(* CoDeSys 2.3 project: drillMachine_NoPackML.pro *)
(* Title: Use of different IEC-61131-3 languages *)
(* Version: 1.0.0 *)
(* Author: Niko Siltala (TUT) *)
(* Description: Use of different IEC-61131-3 languages to control a lift door. *)
(* Libraries: Util.lib 26.9.14 10:12:46, STANDARD.LIB 16.8.17 14:08:57 *)

(* Global variable list: Global_Variables *)
VAR_GLOBAL
	(*Math constants*)
	MATH 				: CONSTANTS_MATH;		(*Mathematical constants from OSCAT 333*)
	lastRandom			: REAL;		(*Last Random number*)

	(*ConveyourIn - Left*)
	I_ConvIn_PartPresent: BOOL;	(*Sensor: Part is present*)
	O_ConvIn_MotON		: BOOL;	(*Conveyour In: Motor ON*)

	(*ConveyourOut - Right*)
	I_ConvOut_PartPresent: BOOL;(*Sensor: Part is present*)
	O_ConvOut_MotON		: BOOL;	(*Conveyour Out: Motor ON*)

	(*Manipulator - Left*)
	I_ManiL_Limit_Up	: BOOL;	(*Manipulator Left: Limit: Up*)
	I_ManiL_Limit_Dn	: BOOL;	(*Manipulator Left: Limit: Down*)
	I_ManiL_Limit_Home	: BOOL;	(*Manipulator Left: Home sensor*)
	I_ManiL_Turned_Left	: BOOL;	(*Manipulator Left: Turned to left*)
	I_ManiL_Turned_Right: BOOL;	(*Manipulator Left: Turned to right*)
	I_ManiL_Gripper_Open: BOOL;	(*Manipulator Left: Gripper is open*)

	O_ManiL_Turn_Left	: BOOL;	(*Manipulator Left: Turn to left position. Controls the valve*)
	O_ManiL_Turn_Right	: BOOL;	(*Manipulator Left: Turn to right position. Controls the valve*)
	O_ManiL_Gripper_Close: BOOL;(*Manipulator Left: Closes Gripper. Controls the valve*)

	bManiL_axZ_Enable	: BOOL;	(*Manipulator Left: Z-axis: enable*)
	bManiL_axZ_Start	: BOOL;	(*Manipulator Left: Z-axis: Start motion*)
	fManiL_axZ_Velo		: REAL;	(*Manipulator Left: Z-axis: Velocity*)
	fManiL_axZ_TargetPos: REAL;	(*Manipulator Left: Z-axis: Target position*)
	fManiL_axZ_CurrPos	: REAL;	(*Manipulator Left: Z-axis: Current position*)
	bManiL_axZ_InTargetPos	: BOOL;	(*Manipulator Left: Z-axis: Target position is reached*)

	(*Drilling Machine*)
	I_Drill_Limit_Up	: BOOL;	(*Drill: Limit: Up*)
	I_Drill_Limit_Dn	: BOOL;	(*Drill: Limit: Down*)
	I_Drill_Limit_Home	: BOOL;	(*Drill: Home sensor*)
	I_Drill_Fixture_Open: BOOL;	(*Drill: Fixture is open*)
	I_Drill_Fixture_Closed: BOOL;	(*Drill: Fixture is closed*)

	O_Drill_Spindle_On	: BOOL;	(*Drill: Turn on drill spindle.*)
	O_Drill_Fixture_Close: BOOL;(*Drill: Closes Fixture. Controls the valve*)

	bDrill_axZ_Enable	: BOOL;	(*Drill: Z-axis: enable*)
	bDrill_axZ_Start	: BOOL;	(*Drill: Z-axis: Start motion*)
	fDrill_axZ_Velo		: REAL;	(*Drill: Z-axis: Velocity*)
	fDrill_axZ_TargetPos: REAL;	(*Drill: Z-axis: Target position*)
	fDrill_axZ_CurrPos	: REAL;	(*Drill: Z-axis: Current position*)
	bDrill_axZ_InTargetPos	: BOOL;	(*Drill: Z-axis: Target position is reached*)

	(*Manipulator - Right*)
	I_ManiR_Limit_Up	: BOOL;	(*Manipulator Right: Limit: Up*)
	I_ManiR_Limit_Dn	: BOOL;	(*Manipulator Right: Limit: Down*)
	I_ManiR_Limit_Home	: BOOL;	(*Manipulator Right: Home sensor*)
	I_ManiR_Turned_Left	: BOOL;	(*Manipulator Right: Turned to left*)
	I_ManiR_Turned_Right: BOOL;	(*Manipulator Right: Turned to right*)
	I_ManiR_Gripper_Open: BOOL;	(*Manipulator Right: Gripper is open*)

	O_ManiR_Turn_Left	: BOOL;	(*Manipulator Right: Turn to left position. Controls the valve*)
	O_ManiR_Turn_Right	: BOOL;	(*Manipulator Right: Turn to right position. Controls the valve*)
	O_ManiR_Gripper_Close: BOOL;(*Manipulator Right: Closes Gripper. Controls the valve*)

	bManiR_axZ_Enable	: BOOL;	(*Manipulator Right: Z-axis: enable*)
	bManiR_axZ_Start	: BOOL;	(*Manipulator Right: Z-axis: Start motion*)
	fManiR_axZ_Velo		: REAL;	(*Manipulator Right: Z-axis: Velocity*)
	fManiR_axZ_TargetPos: REAL;	(*Manipulator Right: Z-axis: Target position*)
	fManiR_axZ_CurrPos	: REAL;	(*Manipulator Right: Z-axis: Current position*)
	bManiR_axZ_InTargetPos	: BOOL;	(*Manipulator Right: Z-axis: Target position is reached*)


	(*Control panel and indications*)
	I_EmergencyClear	: BOOL;	(*Emergency Circuit is clear*)
	I_Btn_Reset		: BOOL;	(*Button: Reset*)
	I_Btn_Start		: BOOL;	(*Button: Start*)
	I_Btn_Stop		: BOOL;	(*Button: Stop*)

	O_Light_Start	: BOOL;	(*Light: Running*)
	O_Light_Stop	: BOOL;	(*Light: Stopped*)
	O_Beacon_Red	: BOOL;	(*Beacon Light: red*)
	O_Beacon_Yellow	: BOOL;	(*Beacon Light: yellow*)
	O_Beacon_Green	: BOOL;	(*Beacon Light: green*)

(* -------------HMI INPUTS (from HMI to PLC) -------------------*)
	HMI_uModeReq		: UINT :=5;		(*Mode request. DEFAULT:PRODUCTION1*)
(* -------------HMI OUTPUTS (from PLC to HMI) -------------------*)
	PLC_uModeCurrent	: UINT;			(*Current Mode*)
	PLC_uStateCurrent	: UINT;			(*Current State*)

(*-----------------------FUNCTION BLOCKS----------------*)
(*	fbStateModel		: FB_PackMLStateModel_ST;	(*FB for executing PackML state model*) *)
END_VAR

(* Data type *)
TYPE CONSTANTS_MATH :
STRUCT
	PI : REAL := 	3.14159265358979323846264338327950288;		(* Kreiszahl PI *)
	PI2 : REAL := 	6.28318530717958647692528676655900576;	(* PI * 2 *)
	PI4 : REAL :=  12.56637061435917295385057353311801152;	(* PI * 4 *)
	PI05 : REAL :=  1.5707963267949;							(* PI / 2 *)
	PI025 : REAL := 0.785398163397448;							(* PI / 4 *)
	PI_INV : REAL := 0.318309886183791;						(* 1 / PI *)
	E : REAL := 	2.71828182845904523536028747135266249;		(* Euler constant e *)
	E_INV : REAL := 0.367879441171442;							(* 1 / e *)
	SQ2 : REAL :=	1.4142135623731;							(* Wurzel von 2 *)
	FACTS : ARRAY[0..12] OF DINT := 1,1,2,6,24,120,720,5040,40320,362880,3628800,39916800,479001600;
END_STRUCT
END_TYPE



(*
From OSCAT 333
revision history
hm	26.10.2008	rev 1.0
	original version

hm	26. mar. 2011	rev 1.1
	added array facts
*)

(* Data type *)
TYPE ST_Part :
(*Data structure for the simulated parts *)
STRUCT
	bExists		: BOOL;	(* Part exists *)
	bHasHole	: BOOL;	(* Part has hole *)
	posX		: REAL;	(* X-position of the part*)
	posY		: REAL;	(* Y-position of the part*)
END_STRUCT
END_TYPE

(* POU PRG_MAIN, ST *)
(* Main Program for Simulated Drill machine.  Perfoms required co-ordination and calling of function blocks
and connects handshake signals etc.  Mode manager FB is used to handle User inputs via HMI
Author: Nicolas Trimborn, nicolas.trimborn@tuni.fi, TUNI
Date: 2020-02-29
Version: 1.0 *) 

PROGRAM PRG_MAIN
VAR
	(* Function Blocks for Machine *)
	fbSFCExample 		: FB_SFC_Example;
	fbMngr					: FB_SimpleManager;
	fbLights				: FB_Lights;
	fbConveyorLeft		: FB_Conveyor_Left;
	fbConveyorRight		: FB_Conveyor_Right;
	fbManipulatorLeft		: FB_Manipulator;
	fbDrill					: FB_Drill;
	fbManipulatorRight	: FB_Manipulator;


	startTrig				: R_TRIG;	 (* Used to restart system after E_Stop Event *)
	(* Status Flags *)
	bStoppedOkAll		: BOOL := TRUE;
	bAll_InitOK			: BOOL := FALSE;

	(* Flags used to handle E_Stop recovery *)
	bStopRequested		: BOOL := FALSE;
	bE_StopRestart		: BOOL := FALSE;

END_VAR
(* Triggers a restart after emergency is cleared *)
startTrig(CLK:= I_EmergencyClear);
IF bAll_InitOK AND NOT bStopRequested THEN
	bE_StopRestart := startTrig.Q;
ELSE
	bE_StopRestart := FALSE;
END_IF

(* Mode Mangager to Handle HMI Buttons*)
fbMngr(
	bEmergencyClear:= I_EmergencyClear,
	bReset:= I_Btn_Reset,
	bStart:= I_Btn_Start OR bE_StopRestart,
	bStop:= I_Btn_Stop,
	bStopOK_All := bStoppedOkAll,
	oEmergencyClear=>,
	oRun=>,
	oStopRequested => bStopRequested );

(* Controls HMI lights based on system state *)
fbLights(
	bReset:= ,
	I_Emergency:= NOT fbMngr.oEmergencyClear,
	I_Stopped:= bStoppedOkAll AND NOT fbMngr.oRun AND fbMngr.oEmergencyClear ,
	I_Stopping:= fbMngr.oEmergencyClear AND NOT fbMngr.oRun AND NOT bStoppedOkAll,
	I_Starting:=  fbMngr.oRun AND NOT bAll_InitOK,
	I_Executing:=  fbMngr.oRun AND bAll_InitOK,
	I_Suspend:= ,
	I_Error:= (PRG_Simulator.wError_ManipL <> 0) OR (PRG_Simulator.wError_ManipR <> 0) OR (PRG_Simulator.wError_Drill <> 0),

	O_Light_Start=> O_Light_Start ,
	O_Light_Stop=> O_Light_Stop ,
	O_Beacon_Red=> O_Beacon_Red,
	O_Beacon_Yellow=> O_Beacon_Yellow,
	O_Beacon_Green=> O_Beacon_Green );

(*Call emergency actions, if emergency is active, other FB not called as long as
Estop is active *)
IF NOT fbMngr.oEmergencyClear THEN
	actEmergency();
	RETURN;
END_IF

(* Continue running system unless all FB indicate ok to Stop *)
IF fbMngr.oRun OR NOT bStoppedOkAll THEN
	fbConveyorLeft (
		bRun := fbMngr.oRun ,
		I_Reset:= NOT  fbMngr.oEmergencyClear  ,
		O_ConvRunning=> O_ConvIn_MotON,
		I_PartEndSensor:=  I_ConvIn_PartPresent,
		hiPartAvail_FromLeft:= TRUE ,
		hiRdyToReceive_FromRight:= fbManipulatorLeft.hoReadyToRecieve_ToLeft,
		hoPartAvail_toRight=> ,
		hoReadyToRecieve_ToLeft=> );
	
	fbManipulatorLeft(
		I_Enable						:=  fbMngr.oRun,
		I_Reset						:=   ,
		b_LeftManip					:= TRUE ,
		I_Mani_Limit_Up				:= I_ManiL_Limit_Up,
		I_Mani_Limit_Dn				:= I_ManiL_Limit_Dn,
		I_Mani_Limit_Home			:= I_ManiL_Limit_Home ,
		I_Mani_Turned_Left			:= I_ManiL_Turned_Left,
		I_Mani_Turned_Right			:= I_ManiL_Turned_Right ,
		I_Mani_Gripper_Open		:= I_ManiL_Gripper_Open ,
		I_fMani_axZ_CurrPos			:= fManiL_axZ_CurrPos ,
		I_bMani_axZ_InTargetPos	:= bManiL_axZ_InTargetPos,
	
		hiPartAvail_FromLeft			:= fbConveyorLeft.hoPartAvail_ToRight ,
		hiRdyToReceive_FromRight	:= fbDrill.hoReadyToRecieve_ToLeft,
		hoReadyToRecieve_ToLeft	=> ,
		hoPartAvail_ToRight			=> ,

		O_Mani_Turn_Left			=> O_ManiL_Turn_Left ,
		O_Mani_Turn_Right			=> O_ManiL_Turn_Right ,
		O_Mani_Gripper_Close		=> O_ManiL_Gripper_Close ,
		O_bMani_axZ_Enable		=> bManiL_axZ_Enable ,
		O_bMani_axZ_Start			=> bManiL_axZ_Start ,
		O_fMani_axZ_Velo			=> fManiL_axZ_Velo,
		O_fMani_axZ_TargetPos		=> fManiL_axZ_TargetPos );
	
	fbDrill(
		I_Enable						:= fbMngr.oRun,
		I_Reset						:=  ,
		I_Drill_Limit_Up				:= I_Drill_Limit_Up,
		I_Drill_Limit_Dn				:= I_Drill_Limit_Dn ,
		I_Drill_Limit_Home			:= I_Drill_Limit_Home,
		I_Drill_Fixture_Open			:= I_Drill_Fixture_Open,
		I_Drill_Fixture_Closed		:= I_Drill_Fixture_Closed,
		fDrill_axZ_CurrPos			:= fDrill_axZ_CurrPos ,
		bDrill_axZ_InTargetPos		:= bDrill_axZ_InTargetPos ,
	
		hiPartAvail_FromLeft			:= fbManipulatorLeft.hoPartAvail_ToRight ,
		hiRdyToReceive_FromRight	:= fbManipulatorRight.hoReadyToRecieve_ToLeft ,
		hoReadyToRecieve_ToLeft	=> ,
		hoPartAvail_ToRight			=> ,
	
		O_Drill_Spindle_On			=> O_Drill_Spindle_On ,
		O_Drill_Fixture_Close		=> O_Drill_Fixture_Close ,
		bDrill_axZ_Enable			=> bDrill_axZ_Enable ,
		bDrill_axZ_Start				=> bDrill_axZ_Start ,
		fDrill_axZ_Velo				=> fDrill_axZ_Velo,
		fDrill_axZ_TargetPos			=> fDrill_axZ_TargetPos );
	
	fbManipulatorRight(
		I_Enable						:=  fbMngr.oRun,
		I_Reset						:=   ,
		b_LeftManip					:= FALSE ,
		I_Mani_Limit_Up				:= I_ManiR_Limit_Up,
		I_Mani_Limit_Dn				:= I_ManiR_Limit_Dn,
		I_Mani_Limit_Home			:= I_ManiR_Limit_Home ,
		I_Mani_Turned_Left			:= I_ManiR_Turned_Left,
		I_Mani_Turned_Right			:= I_ManiR_Turned_Right ,
		I_Mani_Gripper_Open		:= I_ManiR_Gripper_Open ,
		I_fMani_axZ_CurrPos			:= fManiR_axZ_CurrPos ,
		I_bMani_axZ_InTargetPos	:= bManiR_axZ_InTargetPos,
	
		hiPartAvail_FromLeft			:= fbDrill.hoPartAvail_ToRight,
		hiRdyToReceive_FromRight	:= fbConveyorRight.hoReadyToRecieve_ToLeft,
		hoReadyToRecieve_ToLeft	=> ,
		hoPartAvail_ToRight			=> ,
	
		O_Mani_Turn_Left			=> O_ManiR_Turn_Left ,
		O_Mani_Turn_Right			=> O_ManiR_Turn_Right ,
		O_Mani_Gripper_Close		=> O_ManiR_Gripper_Close ,
		O_bMani_axZ_Enable		=> bManiR_axZ_Enable ,
		O_bMani_axZ_Start			=> bManiR_axZ_Start ,
		O_fMani_axZ_Velo			=> fManiR_axZ_Velo,
		O_fMani_axZ_TargetPos		=> fManiR_axZ_TargetPos );
	
	fbConveyorRight (
		bRun := fbMngr.oRun ,
		I_Reset:=   ,
		O_ConvRunning=> O_ConvOut_MotON,
		I_PartEndSensor:=  I_ConvOut_PartPresent,
	
		hiPartAvail_FromLeft:= fbManipulatorRight.hoPartAvail_ToRight  ,
		hiRdyToReceive_FromRight:= TRUE ,
		hoPartAvail_toRight=> ,
		hoReadyToRecieve_ToLeft=> );
END_IF

(* Continously checks if all FB are OK to Stop *)
IF fbConveyorLeft.bStopOk AND fbManipulatorLeft.bStopOk AND fbManipulatorRight.bStopOk AND fbDrill.bStopOk AND  fbConveyorRight.bStopOk THEN
	bStoppedOkAll := TRUE;
ELSE
	bStoppedOkAll := FALSE;
END_IF

(* Checks if all FB are been initialised *)
IF fbManipulatorLeft.bInitialised AND fbManipulatorRight.bInitialised AND fbDrill.bInitialised THEN
	bAll_InitOK := TRUE;
ELSE
	bAll_InitOK := FALSE;
END_IF
END_PROGRAM
ACTION actEmergency:
(* Emergency action which sets outputs to required safe state *)

(* Conveyors *)
O_ConvIn_MotON					:= FALSE;
O_ConvOut_MotON	 			:= FALSE;

(* Manipulators *)
O_ManiL_Turn_Left		 		:= FALSE;
O_ManiL_Turn_Right		 		:= FALSE;
O_ManiR_Turn_Left		 		:= FALSE;
O_ManiR_Turn_Right		 		:= FALSE;
bManiL_axZ_Start					:= FALSE;
bManiR_axZ_Start				:= FALSE;

(*  Avoid Dropping Objects *)
IF I_ManiL_Gripper_Open THEN
	O_ManiL_Gripper_Close 	:= FALSE;
ELSE
	O_ManiL_Gripper_Close		:= TRUE;
END_IF
(* Drill *)
bDrill_axZ_Start 					:= FALSE;
O_Drill_Spindle_On				:= FALSE;

(*  Avoid Toggling fixture Objects *)
IF I_Drill_Fixture_Open THEN
	O_Drill_Fixture_Close 		:= FALSE;
ELSE
	O_Drill_Fixture_Close		:= TRUE;
END_IF
END_ACTION

(* POU Examples/FB_SFC_Example, SFC *)
FUNCTION_BLOCK FB_SFC_Example
VAR_INPUT
	bReset		: BOOL;	(*Reset Request*)
END_VAR
VAR_OUTPUT
END_VAR
VAR
	bLocalReset	: BOOL;	(*Performs local reset*)
	SFCReset 	: BOOL;	(*Resets the execution of SFC to init once this SFCFlag is set true *)
END_VAR
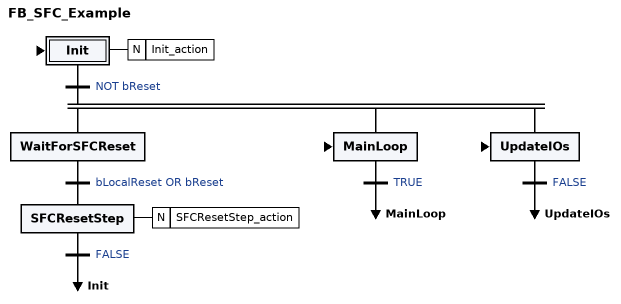
INITIAL_STEP Init:
	Init_action(N);
END_STEP
TRANSITION FROM Init TO (WaitForSFCReset, MainLoop, UpdateIOs) := NOT bReset;
END_TRANSITION
STEP WaitForSFCReset:
END_STEP
TRANSITION FROM WaitForSFCReset TO SFCResetStep := bLocalReset OR bReset;
END_TRANSITION
STEP SFCResetStep:
	SFCResetStep_action(N);
END_STEP
TRANSITION FROM SFCResetStep TO Init := FALSE;
END_TRANSITION
STEP MainLoop:
END_STEP
TRANSITION FROM MainLoop TO MainLoop := TRUE;
END_TRANSITION
STEP UpdateIOs:
END_STEP
TRANSITION FROM UpdateIOs TO UpdateIOs := FALSE;
END_TRANSITION

ACTION Init_action:
SFCReset 	:= FALSE;
bLocalReset	:= FALSE;
END_ACTION

ACTION SFCResetStep_action:
SFCReset := TRUE;
END_ACTION
END_FUNCTION_BLOCK

(* POU FBs/FB_SimpleManager, ST *)
FUNCTION_BLOCK FB_SimpleManager
(*Simple manager following emergency and run/stop state. Outputs can be used to enable user's processes and programs.
Niko Siltala niko.siltala@tuni.fi, 
Tampere University, ENS, ATME.
9.10.2019 v1 *)
VAR_INPUT
	bEmergencyClear		: BOOL;	(*Emergency cleared*)
	bReset				: BOOL;	(*Reset signal*)
	bStart					: BOOL;	(*Start signal*)
	bStop					: BOOL;	(*Stop signal*)
	bStopOK_All			: BOOL;
END_VAR
VAR_OUTPUT
	oEmergencyClear		: BOOL;	(*Emergency is cleared*)
	oRun					: BOOL;	(*System can be started and running*)
	oStopRequested		: BOOL;
END_VAR
VAR
	rsStopRequest		: RS;
	rsEmergency			: RS;
	rsRunning				: RS;
	bResetRequired		: BOOL := TRUE;	(*reset is required*)
END_VAR
(*Defaults*)
(*Reset done*)
IF bReset THEN
	bResetRequired	:= FALSE;
END_IF;

(*Emergency active or cleared?*)
rsEmergency(
	SET:= bReset,
	RESET1:= NOT bEmergencyClear,
	Q1=> oEmergencyClear );

(*Running or stop?*)
rsRunning(
	SET:= bStart,
	RESET1:= (NOT oEmergencyClear) OR bStop OR bResetRequired ,
	Q1=> oRun );

rsStopRequest(
	SET:= bStop,
	RESET1:= bStopOK_All OR bStart,
	Q1=> oStopRequested );
END_FUNCTION_BLOCK

(* POU FBs/FB_Lights, SFC *)
(*Function Block to control the lights of the drill machine based on inputs and functional requirements provided with assignment
Author: Nicolas Trimborn, nicolas.trimborn@tuni.fi, TUNI
Date: 2020-02-29
Version: 1.0 *) 
FUNCTION_BLOCK FB_Lights
VAR_INPUT
	bReset				: BOOL;	(*Reset Request*)
	(* Input States for machine *)
	I_Emergency			: BOOL;
	I_Stopped				: BOOL;
	I_Stopping				: BOOL;
	I_Starting				: BOOL;
	I_Executing			: BOOL;
	I_Suspend			: BOOL;
	I_Error					: BOOL;
END_VAR
VAR_OUTPUT
	(* Light outputs controlled based on input states *)
	O_Light_Start			: BOOL;	(*Light: Running*)
	O_Light_Stop			: BOOL;	(*Light: Stopped*)
	O_Beacon_Red		: BOOL;	(*Beacon Light: red*)
	O_Beacon_Yellow	: BOOL;	(*Beacon Light: yellow*)
	O_Beacon_Green		: BOOL;	(*Beacon Light: greem*)
END_VAR
VAR
	bLocalReset			: BOOL;	(*Performs local reset*)
	SFCReset 			: BOOL;	(*Resets the execution of SFC to init once this SFCFlag is set true *)
 	fbBlinker				: BLINK;     (* Standard Blinker Function Block *)
END_VAR
VAR CONSTANT
	(* 1 Hz Blink requirement *)
	blinkInterval    			: TIME := t#1s;
END_VAR
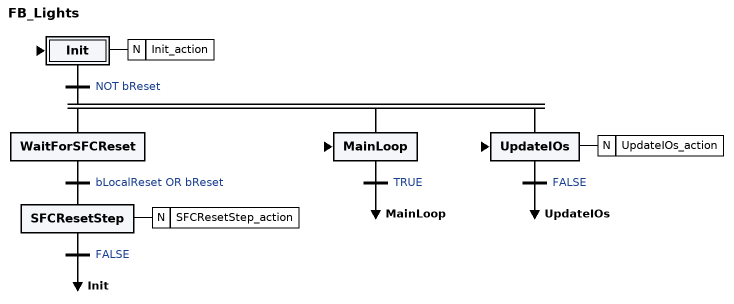
INITIAL_STEP Init:
	Init_action(N);
END_STEP
TRANSITION FROM Init TO (WaitForSFCReset, MainLoop, UpdateIOs) := NOT bReset;
END_TRANSITION
STEP WaitForSFCReset:
END_STEP
TRANSITION FROM WaitForSFCReset TO SFCResetStep := bLocalReset OR bReset;
END_TRANSITION
STEP SFCResetStep:
	SFCResetStep_action(N);
END_STEP
TRANSITION FROM SFCResetStep TO Init := FALSE;
END_TRANSITION
STEP MainLoop:
END_STEP
TRANSITION FROM MainLoop TO MainLoop := TRUE;
END_TRANSITION
STEP UpdateIOs:
	UpdateIOs_action(N);
END_STEP
TRANSITION FROM UpdateIOs TO UpdateIOs := FALSE;
END_TRANSITION

ACTION Init_action:
SFCReset 	:= FALSE;
bLocalReset	:= FALSE;
fbBlinker(ENABLE:= FALSE);
END_ACTION

ACTION SFCResetStep_action:
SFCReset := TRUE;
END_ACTION

ACTION UpdateIOs_action:
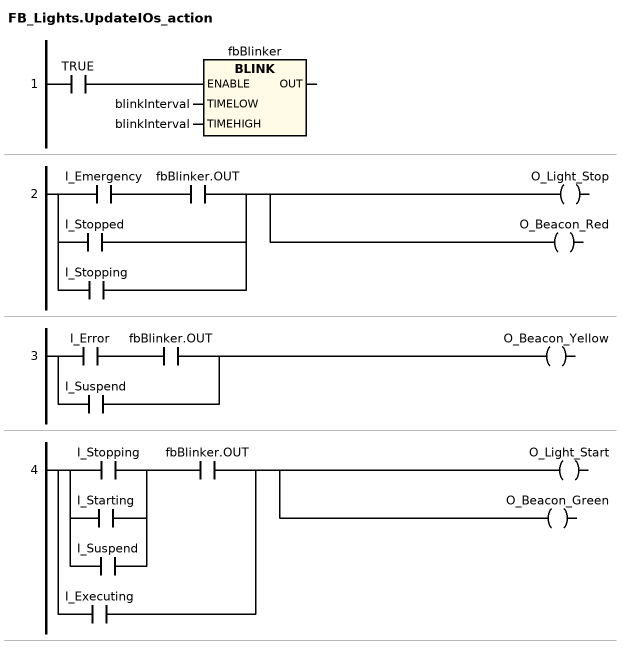
_LD_ (* Ladder Diagram *)
NETWORK 1
	[TRUE] - fbBlinker:BLINK(ENABLE: *, TIMELOW: blinkInterval, TIMEHIGH: blinkInterval)
NETWORK 2
	{ [I_Emergency] - [fbBlinker.OUT] | [I_Stopped] | [I_Stopping] } --- (O_Light_Stop) (O_Beacon_Red)
NETWORK 3
	{ [I_Error] - [fbBlinker.OUT] | [I_Suspend] } --- (O_Beacon_Yellow)
NETWORK 4
	{ { [I_Stopping] | [I_Starting] | [I_Suspend] } - [fbBlinker.OUT] | [I_Executing] } --- (O_Light_Start) (O_Beacon_Green)
_END_LD_
(* the same logic as Structured Text *)
(* Network 1 *)
fbBlinker(ENABLE := TRUE, TIMELOW := blinkInterval, TIMEHIGH := blinkInterval);
(* Network 2 *)
O_Light_Stop := I_Emergency AND fbBlinker.OUT OR I_Stopped OR I_Stopping;
O_Beacon_Red := O_Light_Stop;
(* Network 3 *)
O_Beacon_Yellow := I_Error AND fbBlinker.OUT OR I_Suspend;
(* Network 4 *)
O_Light_Start := (I_Stopping OR I_Starting OR I_Suspend) AND fbBlinker.OUT OR I_Executing;
O_Beacon_Green := O_Light_Start;
END_ACTION
END_FUNCTION_BLOCK

(* POU FBs/FB_Conveyor_Left, SFC *)
(*Function Block to control the left conveyor of simulated drill machine. When bRun is set,
will continously transport added parts to end and notify downstream machine when part is 
availble using SMEMA handshakes.  hiPartAvail_FromLeft always True as this is the start
of production line and assumed to always have parts avalible, but need to be added by operator
Author: Nicolas Trimborn, nicolas.trimborn@tuni.fi, TUNI
Date: 2020-02-29
Version: 1.0 *) 

FUNCTION_BLOCK FB_Conveyor_Left
VAR_INPUT
	bRun		 				: BOOL; 	(*Run Conveyor Function Block*)
	I_Reset		 			: BOOL;	(*Reset Function Block*)
	I_PartEndSensor 			: BOOL;	(*Part End Sensor Input*)

	(* SMEMA Handshake Inputs *)
	hiPartAvail_FromLeft			: BOOL;
	hiRdyToReceive_FromRight	: BOOL;
END_VAR
VAR_OUTPUT
	O_ConvRunning			       : BOOL; (*Output to Simulated conveyor motor*)
	bStopOk						: BOOL; (* bStopOk indicates when there are no parts for processing  and FB is ok to STOP*)

	(* SMEMA Handshake Outputs *)
	hoReadyToRecieve_ToLeft	: BOOL;
	hoPartAvail_ToRight			: BOOL;
END_VAR
VAR
	bLocalReset				: BOOL := FALSE;	(*Performs local reset*)
	SFCReset 				: BOOL := FALSE;	(*Resets the execution of SFC to init once this SFCFlag is set true *)
END_VAR
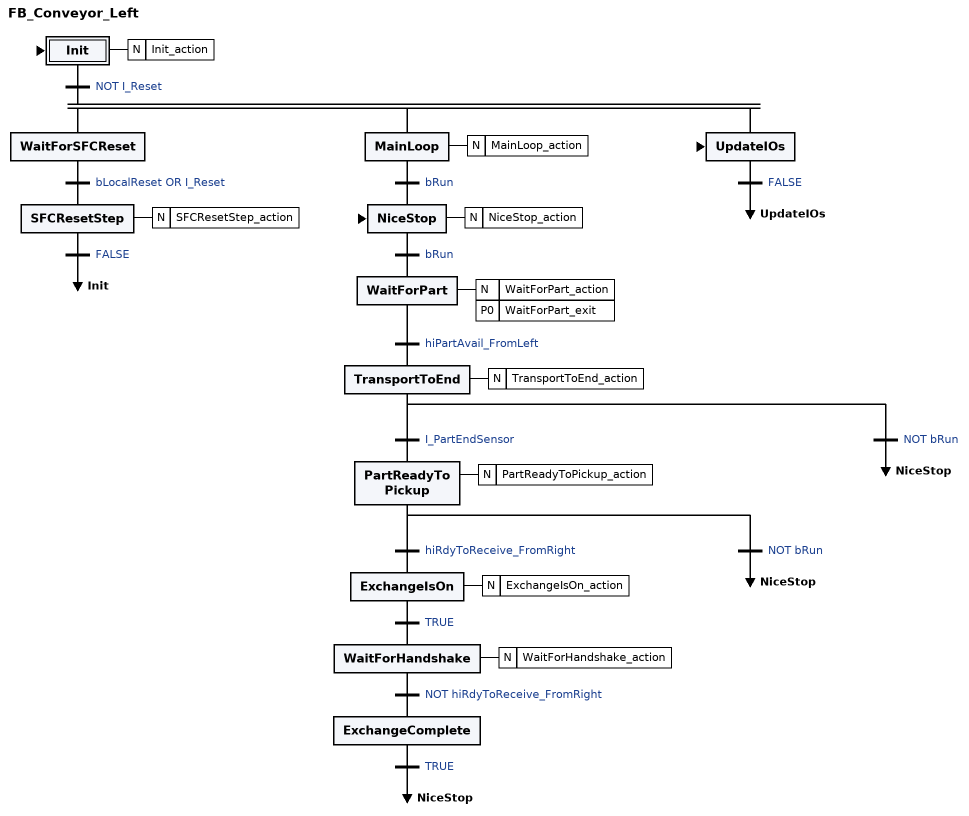
INITIAL_STEP Init:
	Init_action(N);
END_STEP
TRANSITION FROM Init TO (WaitForSFCReset, MainLoop, UpdateIOs) := NOT I_Reset;
END_TRANSITION
STEP WaitForSFCReset:
END_STEP
TRANSITION FROM WaitForSFCReset TO SFCResetStep := bLocalReset OR I_Reset;
END_TRANSITION
STEP MainLoop:
	MainLoop_action(N);
END_STEP
TRANSITION FROM MainLoop TO NiceStop := bRun;
END_TRANSITION
STEP NiceStop:
	NiceStop_action(N);
END_STEP
TRANSITION FROM NiceStop TO WaitForPart := bRun;
END_TRANSITION
STEP WaitForPart:
	WaitForPart_action(N);
	WaitForPart_exit(P0);
END_STEP
TRANSITION FROM WaitForPart TO TransportToEnd := hiPartAvail_FromLeft;
END_TRANSITION
STEP TransportToEnd:
	TransportToEnd_action(N);
END_STEP
TRANSITION FROM TransportToEnd TO PartReadyToPickup := I_PartEndSensor;
END_TRANSITION
TRANSITION FROM TransportToEnd TO NiceStop := NOT bRun;
END_TRANSITION
STEP PartReadyToPickup:
	PartReadyToPickup_action(N);
END_STEP
TRANSITION FROM PartReadyToPickup TO ExchangeIsOn := hiRdyToReceive_FromRight;
END_TRANSITION
TRANSITION FROM PartReadyToPickup TO NiceStop := NOT bRun;
END_TRANSITION
STEP ExchangeIsOn:
	ExchangeIsOn_action(N);
END_STEP
TRANSITION FROM ExchangeIsOn TO WaitForHandshake := TRUE;
END_TRANSITION
STEP WaitForHandshake:
	WaitForHandshake_action(N);
END_STEP
TRANSITION FROM WaitForHandshake TO ExchangeComplete := NOT hiRdyToReceive_FromRight;
END_TRANSITION
STEP ExchangeComplete:
END_STEP
TRANSITION FROM ExchangeComplete TO NiceStop := TRUE;
END_TRANSITION
STEP UpdateIOs:
END_STEP
TRANSITION FROM UpdateIOs TO UpdateIOs := FALSE;
END_TRANSITION
STEP SFCResetStep:
	SFCResetStep_action(N);
END_STEP
TRANSITION FROM SFCResetStep TO Init := FALSE;
END_TRANSITION

ACTION Init_action:
SFCReset := FALSE;
bLocalReset	:= FALSE;
O_ConvRunning := FALSE;
bStopOk := TRUE;
END_ACTION

ACTION MainLoop_action:
hoPartAvail_toRight := FALSE;
END_ACTION

ACTION NiceStop_action:
(* Nice Stop State, FB ok to stop, turn off conveyor and clear Part Avail Flag *)
bStopOk := TRUE;
O_ConvRunning := FALSE;
hoPartAvail_ToRight := FALSE; (* No part availible for downstream manipulator *)
END_ACTION

ACTION WaitForPart_action:
hoReadyToRecieve_ToLeft := TRUE;
END_ACTION

ACTION WaitForPart_exit:
bStopOk := FALSE; (*Part Proccessing *)
END_ACTION

ACTION TransportToEnd_action:
O_ConvRunning := TRUE;
END_ACTION

ACTION PartReadyToPickup_action:
hoPartAvail_ToRight := TRUE; (* Notify downstream machine that part is avalible *)
END_ACTION

ACTION ExchangeIsOn_action:
hoReadyToRecieve_ToLeft := FALSE; (* Proccessing part *)
END_ACTION

ACTION WaitForHandshake_action:
hoPartAvail_ToRight := FALSE; (* Control past to downstream machine *)
END_ACTION

ACTION SFCResetStep_action:
SFCReset := TRUE;
END_ACTION
END_FUNCTION_BLOCK

(* POU FBs/FB_Conveyor_Right, SFC *)
(*Function Block to control the Right conveyor of simulated drill machine. When bRun is set,
and parts are avalible for processing will transport parts deliverd by manipulator to end of 
conveyor to the simulated Stockpile.  

Author: Nicolas Trimborn, nicolas.trimborn@tuni.fi, TUNI
Date: 2020-02-29
Version: 1.0 *) 

FUNCTION_BLOCK FB_Conveyor_Right
VAR_INPUT
	bRun		 				: BOOL; (*Run Conveyor Function Block*)
	I_Reset		 			: BOOL; (*Reset Function Block*)
	I_PartEndSensor 			: BOOL; (*Part End Sensor Input*)

	(* SMEMA Handshake Inputs *)
	hiPartAvail_FromLeft			: BOOL;
	hiRdyToReceive_FromRight	: BOOL;
END_VAR
VAR_OUTPUT
	O_ConvRunning			       : BOOL;  (*Output to Simulated conveyor motor*)
	bStopOk						: BOOL;  (*bStopOk indicates when there are no parts for processing  and FB is ok to STOP*)

	(* SMEMA Handshake Outputs *)
	hoReadyToRecieve_ToLeft	: BOOL;
	hoPartAvail_ToRight			: BOOL;

END_VAR
VAR
	bLocalReset				: BOOL := FALSE;	(*Performs local reset*)
	SFCReset 				: BOOL := FALSE;	(*Resets the execution of SFC to init once this SFCFlag is set true *)
END_VAR
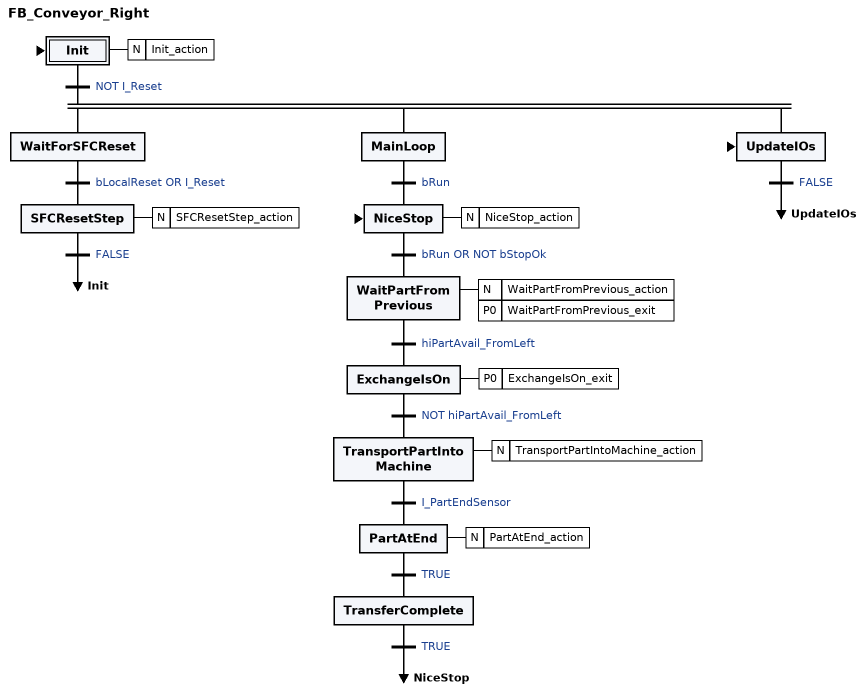
INITIAL_STEP Init:
	Init_action(N);
END_STEP
TRANSITION FROM Init TO (WaitForSFCReset, MainLoop, UpdateIOs) := NOT I_Reset;
END_TRANSITION
STEP WaitForSFCReset:
END_STEP
TRANSITION FROM WaitForSFCReset TO SFCResetStep := bLocalReset OR I_Reset;
END_TRANSITION
STEP MainLoop:
END_STEP
TRANSITION FROM MainLoop TO NiceStop := bRun;
END_TRANSITION
STEP NiceStop:
	NiceStop_action(N);
END_STEP
TRANSITION FROM NiceStop TO WaitPartFromPrevious := bRun OR NOT bStopOk;
END_TRANSITION
STEP WaitPartFromPrevious:
	WaitPartFromPrevious_action(N);
	WaitPartFromPrevious_exit(P0);
END_STEP
TRANSITION FROM WaitPartFromPrevious TO ExchangeIsOn := hiPartAvail_FromLeft;
END_TRANSITION
STEP ExchangeIsOn:
	ExchangeIsOn_exit(P0);
END_STEP
TRANSITION FROM ExchangeIsOn TO TransportPartIntoMachine := NOT hiPartAvail_FromLeft;
END_TRANSITION
STEP TransportPartIntoMachine:
	TransportPartIntoMachine_action(N);
END_STEP
TRANSITION FROM TransportPartIntoMachine TO PartAtEnd := I_PartEndSensor;
END_TRANSITION
STEP PartAtEnd:
	PartAtEnd_action(N);
END_STEP
TRANSITION FROM PartAtEnd TO TransferComplete := TRUE;
END_TRANSITION
STEP TransferComplete:
END_STEP
TRANSITION FROM TransferComplete TO NiceStop := TRUE;
END_TRANSITION
STEP UpdateIOs:
END_STEP
TRANSITION FROM UpdateIOs TO UpdateIOs := FALSE;
END_TRANSITION
STEP SFCResetStep:
	SFCResetStep_action(N);
END_STEP
TRANSITION FROM SFCResetStep TO Init := FALSE;
END_TRANSITION

ACTION Init_action:
SFCReset := FALSE;
bLocalReset	:= FALSE;
O_ConvRunning := FALSE;
bStopOK						:= TRUE;
END_ACTION

ACTION NiceStop_action:
(* Ok To stop if there are no parts pending from Adjacent manipulator *)
IF hiPartAvail_FromLeft THEN
	bStopOk := FALSE;
ELSE
	bStopOk := TRUE;
END_IF
END_ACTION

ACTION WaitPartFromPrevious_action:
(* Set SMEMA flags to recieve part*)
hoReadyToRecieve_ToLeft := TRUE;
hoPartAvail_toRight := FALSE;
END_ACTION

ACTION WaitPartFromPrevious_exit:
bStopOK	:= FALSE;
END_ACTION

ACTION ExchangeIsOn_exit:
O_ConvRunning := FALSE;
END_ACTION

ACTION TransportPartIntoMachine_action:
(* Move Part to end *)
O_ConvRunning := TRUE;
(* Handshake to indicate part is not under conveyor control *)
hoReadyToRecieve_ToLeft := FALSE;
END_ACTION

ACTION PartAtEnd_action:
(* Stop conveyor when part reaches end *)
O_ConvRunning := FALSE;
hoPartAvail_ToRight := TRUE;
END_ACTION

ACTION SFCResetStep_action:
SFCReset := TRUE;
END_ACTION
END_FUNCTION_BLOCK

(* POU FBs/FB_Manipulator, SFC *)
(*Function Block to control both manipulators of simulated drill machine. When I_Enable is set,
will execute a movement sequence based on Handshakes recieved from adjacent machines. When 
parts are avalible for collection and when they have been delivered and recieved successfully.
bLeftManip Flag is used to determine if left of right manipulator to determine pick and place heights etc.  
Author: Nicolas Trimborn, nicolas.trimborn@tuni.fi, TUNI
Date: 2020-02-29
Version: 1.0 *) 

FUNCTION_BLOCK FB_Manipulator
VAR_INPUT
	I_Enable		 				: BOOL; (*Run Manipulator Function Block*)
	I_Reset		 				: BOOL; (*Reset Function Block*)
	b_LeftManip					: BOOL; (*Flag to indicate if this is Left Manip*)

	(* SMEMA Handshake Inputs *)
	hiPartAvail_FromLeft			: BOOL;
	hiRdyToReceive_FromRight	: BOOL;

	(* Manipulator Sensor *)
	I_Mani_Limit_Up				: BOOL;	(*Manipulator Left: Limit: Up*)
	I_Mani_Limit_Dn				: BOOL;	(*Manipulator Left: Limit: Down*)
	I_Mani_Limit_Home			: BOOL;	(*Manipulator Left: Home sensor*)
	I_Mani_Turned_Left			: BOOL;	(*Manipulator Left: Turned to left*)
	I_Mani_Turned_Right			: BOOL;	(*Manipulator Left: Turned to right*)
	I_Mani_Gripper_Open		: BOOL;	(*Manipulator Left: Gripper is open*)

	(* Manipulator Controls *)
	I_fMani_axZ_CurrPos			: REAL;	(*Manipulator Left: Z-axis: Current position*)
	I_bMani_axZ_InTargetPos	: BOOL;	(*Manipulator Left: Z-axis: Target position is reached*)

END_VAR
VAR_OUTPUT
	bInitialised					: BOOL; 	(*Initialisation complete flag *)
	bStopOk						: BOOL;      (* bStopOk indicates when there are no parts for processing  and FB is ok to STOP*)

	(* SMEMA Handshake Outputs *)
	hoReadyToRecieve_ToLeft	: BOOL;
	hoPartAvail_ToRight			: BOOL;

	(* Manipulator Outputs *)
	O_Mani_Turn_Left			: BOOL;	(*Manipulator Left: Turn to left position. Controls the valve*)
	O_Mani_Turn_Right			: BOOL;	(*Manipulator Left: Turn to right position. Controls the valve*)
	O_Mani_Gripper_Close		: BOOL;	(*Manipulator Left: Closes Gripper. Controls the valve*)

	(* Manipulator Z axis Control *)
	O_bMani_axZ_Enable		: BOOL;	(*Manipulator Left: Z-axis: enable*)
	O_bMani_axZ_Start			: BOOL;	(*Manipulator Left: Z-axis: Start motion*)
	O_fMani_axZ_Velo			: REAL;	(*Manipulator Left: Z-axis: Velocity*)
	O_fMani_axZ_TargetPos		: REAL;	(*Manipulator Left: Z-axis: Target position*)


END_VAR
VAR
	(* Pick/Place sequence flags *)
	bPick						: BOOL := FALSE;
	bPicked					: BOOL := FALSE;
	bPlace						: BOOL := FALSE;
	bPlaced					: BOOL := FALSE;

	bManipulatorHomed		: BOOL := FALSE; (* Homing Completed Flag, only need on startup*)

	(*Timer and delay for Z axis motion block to give time for block to perform motion and clear/set flags *)
	tonMoveDelay				: TON;
	tMoveDelay				: TIME := T#1s;

	bLocalReset				: BOOL := FALSE;	(*Performs local reset*)
	SFCReset 				: BOOL := FALSE;	(*Resets the execution of SFC to init once this SFCFlag is set true *)
END_VAR
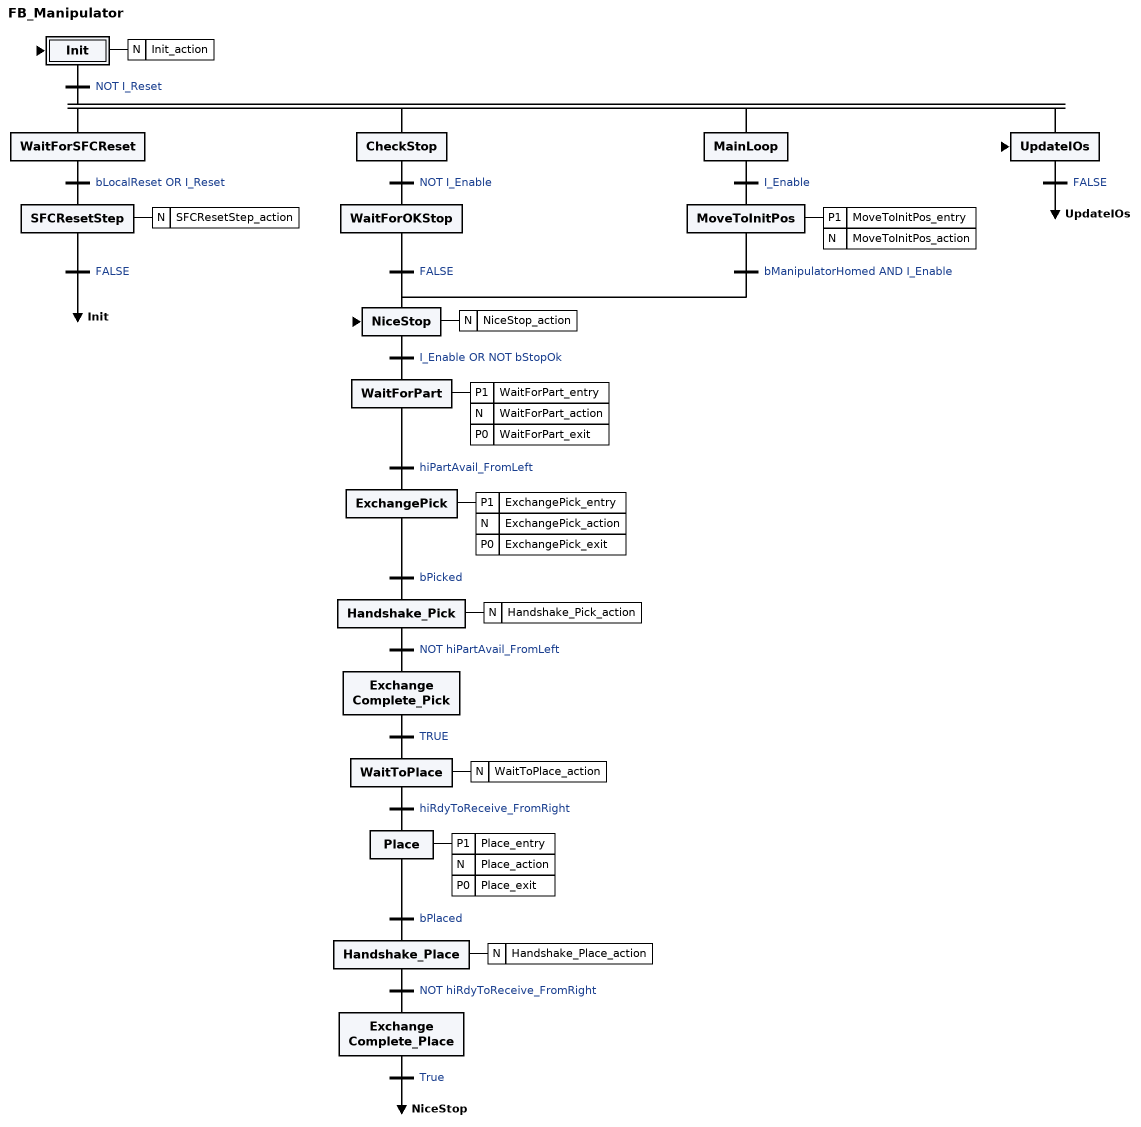
INITIAL_STEP Init:
	Init_action(N);
END_STEP
TRANSITION FROM Init TO (WaitForSFCReset, CheckStop, MainLoop, UpdateIOs) := NOT I_Reset;
END_TRANSITION
STEP WaitForSFCReset:
END_STEP
TRANSITION FROM WaitForSFCReset TO SFCResetStep := bLocalReset OR I_Reset;
END_TRANSITION
STEP CheckStop:
END_STEP
TRANSITION FROM CheckStop TO WaitForOKStop := NOT I_Enable;
END_TRANSITION
STEP WaitForOKStop:
END_STEP
TRANSITION FROM WaitForOKStop TO NiceStop := FALSE;
END_TRANSITION
STEP MainLoop:
END_STEP
TRANSITION FROM MainLoop TO MoveToInitPos := I_Enable;
END_TRANSITION
STEP MoveToInitPos:
	MoveToInitPos_entry(P1);
	MoveToInitPos_action(N);
END_STEP
TRANSITION FROM MoveToInitPos TO NiceStop := bManipulatorHomed AND I_Enable;
END_TRANSITION
STEP NiceStop:
	NiceStop_action(N);
END_STEP
TRANSITION FROM NiceStop TO WaitForPart := I_Enable OR NOT bStopOk;
END_TRANSITION
STEP WaitForPart:
	WaitForPart_entry(P1);
	WaitForPart_action(N);
	WaitForPart_exit(P0);
END_STEP
TRANSITION FROM WaitForPart TO ExchangePick := hiPartAvail_FromLeft;
END_TRANSITION
STEP ExchangePick:
	ExchangePick_entry(P1);
	ExchangePick_action(N);
	ExchangePick_exit(P0);
END_STEP
TRANSITION FROM ExchangePick TO Handshake_Pick := bPicked;
END_TRANSITION
STEP Handshake_Pick:
	Handshake_Pick_action(N);
END_STEP
TRANSITION FROM Handshake_Pick TO ExchangeComplete_Pick := NOT hiPartAvail_FromLeft;
END_TRANSITION
STEP ExchangeComplete_Pick:
END_STEP
TRANSITION FROM ExchangeComplete_Pick TO WaitToPlace := TRUE;
END_TRANSITION
STEP WaitToPlace:
	WaitToPlace_action(N);
END_STEP
TRANSITION FROM WaitToPlace TO Place := hiRdyToReceive_FromRight;
END_TRANSITION
STEP Place:
	Place_entry(P1);
	Place_action(N);
	Place_exit(P0);
END_STEP
TRANSITION FROM Place TO Handshake_Place := bPlaced;
END_TRANSITION
STEP Handshake_Place:
	Handshake_Place_action(N);
END_STEP
TRANSITION FROM Handshake_Place TO ExchangeComplete_Place := NOT hiRdyToReceive_FromRight;
END_TRANSITION
STEP ExchangeComplete_Place:
END_STEP
TRANSITION FROM ExchangeComplete_Place TO NiceStop := True;
END_TRANSITION
STEP UpdateIOs:
END_STEP
TRANSITION FROM UpdateIOs TO UpdateIOs := FALSE;
END_TRANSITION
STEP SFCResetStep:
	SFCResetStep_action(N);
END_STEP
TRANSITION FROM SFCResetStep TO Init := FALSE;
END_TRANSITION

ACTION Init_action:
(* State Flags *)
bManipulatorHomed 			:= FALSE;
bStopOK						:= TRUE;

(* Reset Flags *)
SFCReset 					:= FALSE;
bLocalReset					:= FALSE;

(* Init Handshakes *)
hoReadyToRecieve_ToLeft	:= FALSE;
hoPartAvail_ToRight			:= FALSE;
END_ACTION

ACTION MoveToInitPos_entry:
bStopOk := FALSE;
END_ACTION

ACTION MoveToInitPos_action:
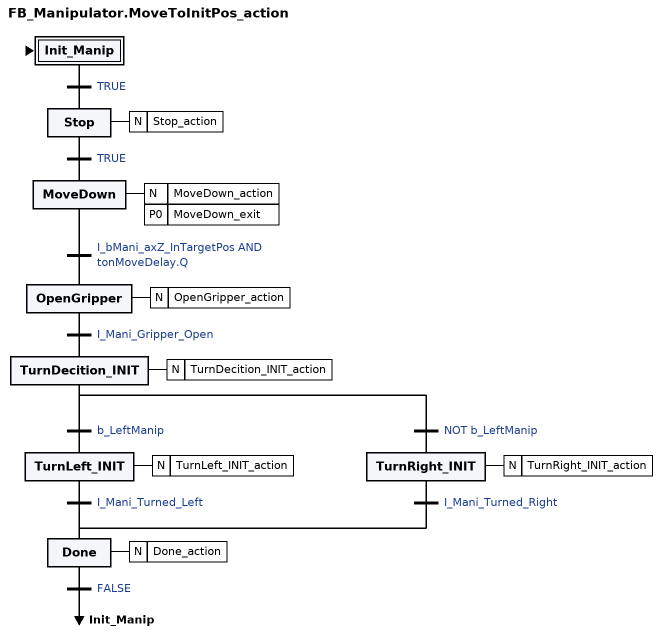
INITIAL_STEP Init_Manip:
END_STEP
TRANSITION FROM Init_Manip TO Stop := TRUE;
END_TRANSITION
STEP Stop:
	Stop_action(N);
END_STEP
TRANSITION FROM Stop TO MoveDown := TRUE;
END_TRANSITION
STEP MoveDown:
	MoveDown_action(N);
	MoveDown_exit(P0);
END_STEP
TRANSITION FROM MoveDown TO OpenGripper := I_bMani_axZ_InTargetPos AND tonMoveDelay.Q;
END_TRANSITION
STEP OpenGripper:
	OpenGripper_action(N);
END_STEP
TRANSITION FROM OpenGripper TO TurnDecition_INIT := I_Mani_Gripper_Open;
END_TRANSITION
STEP TurnDecition_INIT:
	TurnDecition_INIT_action(N);
END_STEP
TRANSITION FROM TurnDecition_INIT TO TurnLeft_INIT := b_LeftManip;
END_TRANSITION
TRANSITION FROM TurnDecition_INIT TO TurnRight_INIT := NOT b_LeftManip;
END_TRANSITION
STEP TurnLeft_INIT:
	TurnLeft_INIT_action(N);
END_STEP
TRANSITION FROM TurnLeft_INIT TO Done := I_Mani_Turned_Left;
END_TRANSITION
STEP TurnRight_INIT:
	TurnRight_INIT_action(N);
END_STEP
TRANSITION FROM TurnRight_INIT TO Done := I_Mani_Turned_Right;
END_TRANSITION
STEP Done:
	Done_action(N);
END_STEP
TRANSITION FROM Done TO Init_Manip := FALSE;
END_TRANSITION

ACTION Stop_action:
O_fMani_axZ_Velo		:= 0;
O_Mani_Turn_Left		:= FALSE;
O_Mani_Turn_Right		:= FALSE;
END_ACTION

ACTION MoveDown_action:
O_bMani_axZ_Enable		:= TRUE;
O_fMani_axZ_Velo			:= 5;
O_fMani_axZ_TargetPos		:= -43;
O_bMani_axZ_Start			:= TRUE;
(* Start Movement Timer *)
tonMoveDelay(IN:=TRUE , PT:= tMoveDelay);
END_ACTION

ACTION MoveDown_exit:
(* Reset movement timer *)
tonMoveDelay(IN:=FALSE);
(* Reset Start Flag *)
O_bMani_axZ_Start	:= FALSE;
END_ACTION

ACTION OpenGripper_action:
O_Mani_Gripper_Close := FALSE;
END_ACTION

ACTION TurnDecition_INIT_action:
IF b_LeftManip THEN
	O_Mani_Turn_Right 	 := TRUE;
	O_Mani_Turn_Left 	 := FALSE;
ELSE
	O_Mani_Turn_Right	 := FALSE;
	O_Mani_Turn_Left 	 := TRUE;
END_IF
END_ACTION

ACTION TurnLeft_INIT_action:
O_Mani_Turn_Right 	 := FALSE;
O_Mani_Turn_Left 	 := TRUE;
END_ACTION

ACTION TurnRight_INIT_action:
O_Mani_Turn_Right 	 := TRUE;
O_Mani_Turn_Left 	 := FALSE;
END_ACTION

ACTION Done_action:
bManipulatorHomed := TRUE;
bInitialised  := TRUE;
END_ACTION
END_ACTION

ACTION NiceStop_action:
(* Ok To stop if there are no parts pending from Adjacent Machine *)
IF hiPartAvail_FromLeft THEN
	bStopOk := FALSE;
ELSE
	bStopOk := TRUE;
END_IF
END_ACTION

ACTION WaitForPart_entry:
bPicked := FALSE;
bPlaced := FALSE;
END_ACTION

ACTION WaitForPart_action:
(* Set ready to recieve flag for upstream machines *)
hoReadyToRecieve_ToLeft	 := TRUE;
END_ACTION

ACTION WaitForPart_exit:
(* Starting Sequence, not ok to stop *)
bStopOK	:= FALSE;
END_ACTION

ACTION ExchangePick_entry:
bPick := TRUE;
END_ACTION

ACTION ExchangePick_action:
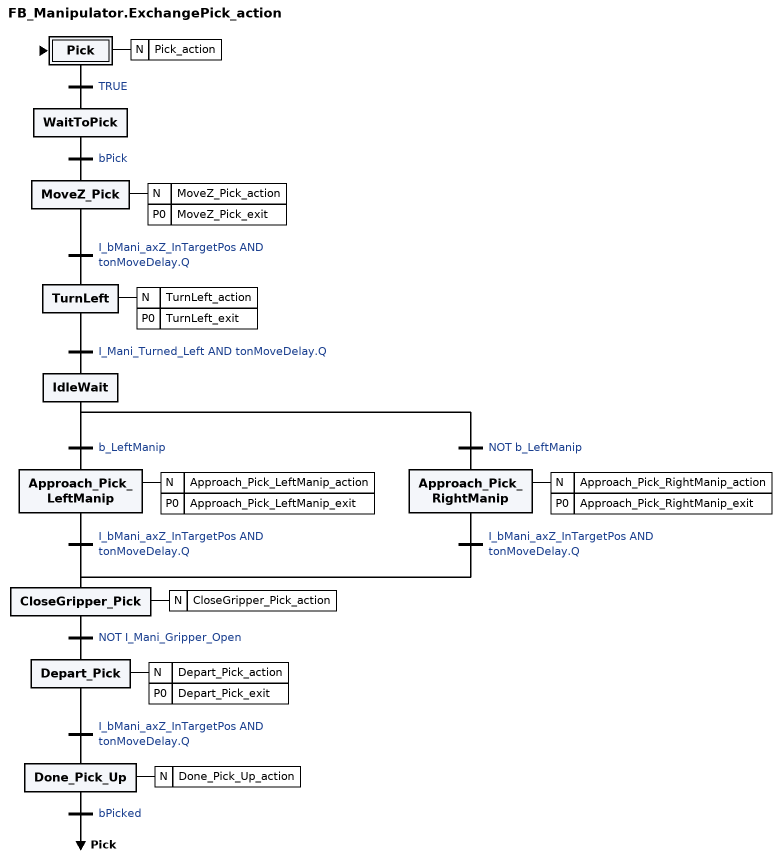
INITIAL_STEP Pick:
	Pick_action(N);
END_STEP
TRANSITION FROM Pick TO WaitToPick := TRUE;
END_TRANSITION
STEP WaitToPick:
END_STEP
TRANSITION FROM WaitToPick TO MoveZ_Pick := bPick;
END_TRANSITION
STEP MoveZ_Pick:
	MoveZ_Pick_action(N);
	MoveZ_Pick_exit(P0);
END_STEP
TRANSITION FROM MoveZ_Pick TO TurnLeft := I_bMani_axZ_InTargetPos AND tonMoveDelay.Q;
END_TRANSITION
STEP TurnLeft:
	TurnLeft_action(N);
	TurnLeft_exit(P0);
END_STEP
TRANSITION FROM TurnLeft TO IdleWait := I_Mani_Turned_Left AND tonMoveDelay.Q;
END_TRANSITION
STEP IdleWait:
END_STEP
TRANSITION FROM IdleWait TO Approach_Pick_LeftManip := b_LeftManip;
END_TRANSITION
TRANSITION FROM IdleWait TO Approach_Pick_RightManip := NOT b_LeftManip;
END_TRANSITION
STEP Approach_Pick_LeftManip:
	Approach_Pick_LeftManip_action(N);
	Approach_Pick_LeftManip_exit(P0);
END_STEP
TRANSITION FROM Approach_Pick_LeftManip TO CloseGripper_Pick := I_bMani_axZ_InTargetPos AND tonMoveDelay.Q;
END_TRANSITION
STEP Approach_Pick_RightManip:
	Approach_Pick_RightManip_action(N);
	Approach_Pick_RightManip_exit(P0);
END_STEP
TRANSITION FROM Approach_Pick_RightManip TO CloseGripper_Pick := I_bMani_axZ_InTargetPos AND tonMoveDelay.Q;
END_TRANSITION
STEP CloseGripper_Pick:
	CloseGripper_Pick_action(N);
END_STEP
TRANSITION FROM CloseGripper_Pick TO Depart_Pick := NOT I_Mani_Gripper_Open;
END_TRANSITION
STEP Depart_Pick:
	Depart_Pick_action(N);
	Depart_Pick_exit(P0);
END_STEP
TRANSITION FROM Depart_Pick TO Done_Pick_Up := I_bMani_axZ_InTargetPos AND tonMoveDelay.Q;
END_TRANSITION
STEP Done_Pick_Up:
	Done_Pick_Up_action(N);
END_STEP
TRANSITION FROM Done_Pick_Up TO Pick := bPicked;
END_TRANSITION

ACTION Pick_action:
bPicked := FALSE;
END_ACTION

ACTION MoveZ_Pick_action:
O_bMani_axZ_Enable := TRUE;
tonMoveDelay(IN:=TRUE , PT:= tMoveDelay);
O_fMani_axZ_Velo :=10;
O_fMani_axZ_TargetPos := -45;
O_bMani_axZ_Start := TRUE;
END_ACTION

ACTION MoveZ_Pick_exit:
tonMoveDelay(IN:=FALSE );
O_bMani_axZ_Start := FALSE;
END_ACTION

ACTION TurnLeft_action:
tonMoveDelay(IN:=TRUE , PT:= tMoveDelay);
O_Mani_Turn_Left 	 := TRUE;
O_Mani_Turn_Right 	 := FALSE;
END_ACTION

ACTION TurnLeft_exit:
tonMoveDelay(IN:=FALSE);
END_ACTION

ACTION Approach_Pick_LeftManip_action:
bPicked := FALSE;
tonMoveDelay(IN:=TRUE , PT:= tMoveDelay);
O_fMani_axZ_Velo :=10;
O_fMani_axZ_TargetPos := -120;
O_bMani_axZ_Start := TRUE;
END_ACTION

ACTION Approach_Pick_LeftManip_exit:
(*Clear flags *)
O_bMani_axZ_Start := FALSE;
tonMoveDelay(IN:=FALSE);
END_ACTION

ACTION Approach_Pick_RightManip_action:
bPicked := FALSE;
tonMoveDelay(IN:=TRUE , PT:= tMoveDelay);
O_fMani_axZ_Velo :=10;
O_fMani_axZ_TargetPos := -74;
O_bMani_axZ_Start := TRUE;
END_ACTION

ACTION Approach_Pick_RightManip_exit:
(*Clear flags *)
O_bMani_axZ_Start := FALSE;
tonMoveDelay(IN:=FALSE);
END_ACTION

ACTION CloseGripper_Pick_action:
O_Mani_Gripper_Close := TRUE;
END_ACTION

ACTION Depart_Pick_action:
O_fMani_axZ_Velo :=10;
O_fMani_axZ_TargetPos := -45;
O_bMani_axZ_Start := TRUE;
tonMoveDelay(IN:=TRUE , PT:= tMoveDelay);
END_ACTION

ACTION Depart_Pick_exit:
O_bMani_axZ_Start := FALSE;
tonMoveDelay(IN:=FALSE);
END_ACTION

ACTION Done_Pick_Up_action:
(* Sequeance completed*)
bPick		 := FALSE;
bPicked	 := TRUE;
END_ACTION
END_ACTION

ACTION ExchangePick_exit:
bPick := FALSE;
bPlaced := FALSE;
END_ACTION

ACTION Handshake_Pick_action:
(* Signal Upstream that part has been picked *)
hoReadyToRecieve_ToLeft := FALSE;
END_ACTION

ACTION WaitToPlace_action:
(*Notify downstream that there is a part ready to place *)
hoPartAvail_ToRight := TRUE;
END_ACTION

ACTION Place_entry:
bPlace   := TRUE;
bPicked := FALSE;
END_ACTION

ACTION Place_action:
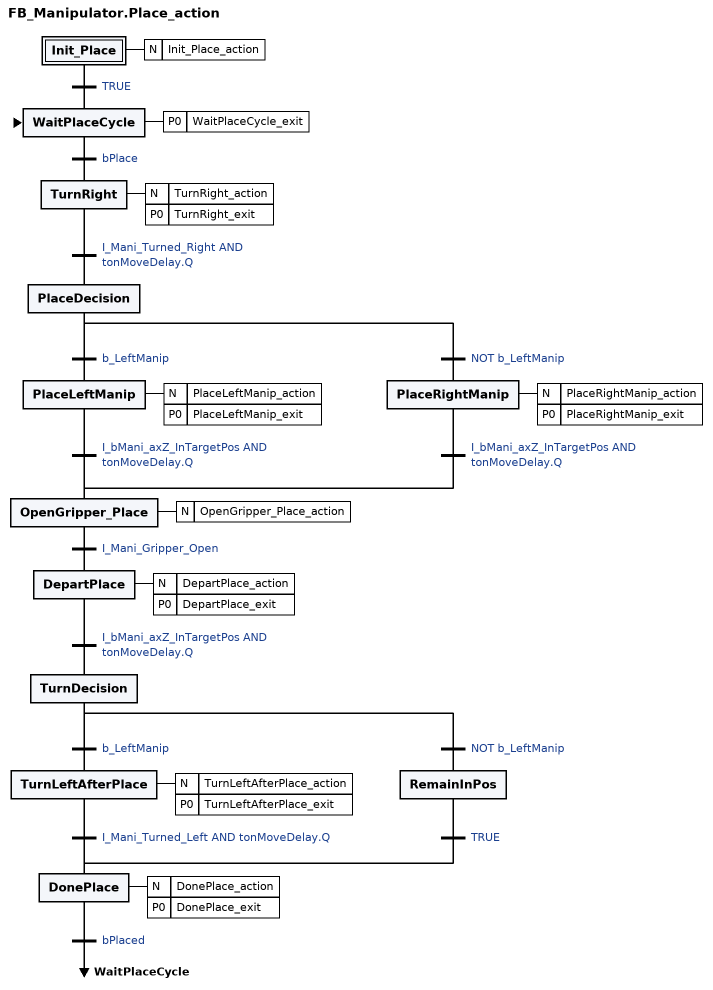
INITIAL_STEP Init_Place:
	Init_Place_action(N);
END_STEP
TRANSITION FROM Init_Place TO WaitPlaceCycle := TRUE;
END_TRANSITION
STEP WaitPlaceCycle:
	WaitPlaceCycle_exit(P0);
END_STEP
TRANSITION FROM WaitPlaceCycle TO TurnRight := bPlace;
END_TRANSITION
STEP TurnRight:
	TurnRight_action(N);
	TurnRight_exit(P0);
END_STEP
TRANSITION FROM TurnRight TO PlaceDecision := I_Mani_Turned_Right AND tonMoveDelay.Q;
END_TRANSITION
STEP PlaceDecision:
END_STEP
TRANSITION FROM PlaceDecision TO PlaceLeftManip := b_LeftManip;
END_TRANSITION
TRANSITION FROM PlaceDecision TO PlaceRightManip := NOT b_LeftManip;
END_TRANSITION
STEP PlaceLeftManip:
	PlaceLeftManip_action(N);
	PlaceLeftManip_exit(P0);
END_STEP
TRANSITION FROM PlaceLeftManip TO OpenGripper_Place := I_bMani_axZ_InTargetPos AND tonMoveDelay.Q;
END_TRANSITION
STEP PlaceRightManip:
	PlaceRightManip_action(N);
	PlaceRightManip_exit(P0);
END_STEP
TRANSITION FROM PlaceRightManip TO OpenGripper_Place := I_bMani_axZ_InTargetPos AND tonMoveDelay.Q;
END_TRANSITION
STEP OpenGripper_Place:
	OpenGripper_Place_action(N);
END_STEP
TRANSITION FROM OpenGripper_Place TO DepartPlace := I_Mani_Gripper_Open;
END_TRANSITION
STEP DepartPlace:
	DepartPlace_action(N);
	DepartPlace_exit(P0);
END_STEP
TRANSITION FROM DepartPlace TO TurnDecision := I_bMani_axZ_InTargetPos AND tonMoveDelay.Q;
END_TRANSITION
STEP TurnDecision:
END_STEP
TRANSITION FROM TurnDecision TO TurnLeftAfterPlace := b_LeftManip;
END_TRANSITION
TRANSITION FROM TurnDecision TO RemainInPos := NOT b_LeftManip;
END_TRANSITION
STEP TurnLeftAfterPlace:
	TurnLeftAfterPlace_action(N);
	TurnLeftAfterPlace_exit(P0);
END_STEP
TRANSITION FROM TurnLeftAfterPlace TO DonePlace := I_Mani_Turned_Left AND tonMoveDelay.Q;
END_TRANSITION
STEP RemainInPos:
END_STEP
TRANSITION FROM RemainInPos TO DonePlace := TRUE;
END_TRANSITION
STEP DonePlace:
	DonePlace_action(N);
	DonePlace_exit(P0);
END_STEP
TRANSITION FROM DonePlace TO WaitPlaceCycle := bPlaced;
END_TRANSITION

ACTION Init_Place_action:
bPlaced := FALSE;
END_ACTION

ACTION WaitPlaceCycle_exit:
bPlaced := FALSE;
END_ACTION

ACTION TurnRight_action:
tonMoveDelay(IN:=TRUE , PT:= tMoveDelay);
O_Mani_Turn_Right	 := TRUE;
O_Mani_Turn_Left 	 := FALSE;
END_ACTION

ACTION TurnRight_exit:
tonMoveDelay(IN:=FALSE);
END_ACTION

ACTION PlaceLeftManip_action:
tonMoveDelay(IN:=TRUE , PT:= tMoveDelay);
O_fMani_axZ_Velo :=10;
O_fMani_axZ_TargetPos := -74;
O_bMani_axZ_Start := TRUE;
END_ACTION

ACTION PlaceLeftManip_exit:
O_bMani_axZ_Start 	:= FALSE;
tonMoveDelay(IN		:=FALSE);
END_ACTION

ACTION PlaceRightManip_action:
tonMoveDelay(IN:=TRUE , PT:= tMoveDelay);
O_fMani_axZ_Velo :=10;
O_fMani_axZ_TargetPos := -120;
O_bMani_axZ_Start := TRUE;
END_ACTION

ACTION PlaceRightManip_exit:
O_bMani_axZ_Start := FALSE;
tonMoveDelay(IN:=FALSE);
END_ACTION

ACTION OpenGripper_Place_action:
O_Mani_Gripper_Close := FALSE;
END_ACTION

ACTION DepartPlace_action:
tonMoveDelay(IN:=TRUE , PT:= tMoveDelay);
O_fMani_axZ_Velo :=5;
O_fMani_axZ_TargetPos := -40;
O_bMani_axZ_Start := TRUE;
END_ACTION

ACTION DepartPlace_exit:
(* Reset Flags and blocks *)
O_bMani_axZ_Start := FALSE;
tonMoveDelay(IN:=FALSE);
END_ACTION

ACTION TurnLeftAfterPlace_action:
tonMoveDelay(IN:=TRUE , PT:= tMoveDelay);
O_Mani_Turn_Right	 := FALSE;
O_Mani_Turn_Left 	 := TRUE;
END_ACTION

ACTION TurnLeftAfterPlace_exit:
tonMoveDelay(IN:=FALSE);
END_ACTION

ACTION DonePlace_action:
bPlaced				:= TRUE;
END_ACTION

ACTION DonePlace_exit:
bPlaced := FALSE;
END_ACTION
END_ACTION

ACTION Place_exit:
bPlace := FALSE;
bPicked := FALSE;
END_ACTION

ACTION Handshake_Place_action:
hoPartAvail_ToRight := FALSE;
END_ACTION

ACTION SFCResetStep_action:
SFCReset := TRUE;
END_ACTION
END_FUNCTION_BLOCK

(* POU FBs/FB_Drill, SFC *)
(*Function Block to control the Drill of simulated drill machine. When I_Enable is set,
will execute a drilling sequence on parts delivered and retreieved by adjacent manipulators.
Handshakes are used to indicate when drill is avalible for new parts and when completed
parts can be collected
Author: Nicolas Trimborn, nicolas.trimborn@tuni.fi, TUNI
Date: 2020-02-29
Version: 1.0 *) 

FUNCTION_BLOCK FB_Drill
VAR_INPUT
	I_Enable		 				: BOOL; (*Run Drill Function Block*)
	I_Reset						: BOOL; (*Reset Function Block*)
	(* Drill Sensor *)
	I_Drill_Limit_Up				: BOOL;	(*Drill: Limit: Up*)
	I_Drill_Limit_Dn				: BOOL;	(*Drill: Limit: Down*)
	I_Drill_Limit_Home			: BOOL;	(*Drill: Home sensor*)
	I_Drill_Fixture_Open			: BOOL;	(*Drill: Fixture is open*)
	I_Drill_Fixture_Closed		: BOOL;	(*Drill: Fixture is closed*)

	(* Drill Z Axis Feedback *)
	fDrill_axZ_CurrPos			: REAL;	(*Drill: Z-axis: Current position*)
	bDrill_axZ_InTargetPos		: BOOL;	(*Drill: Z-axis: Target position is reached*)

	(* SMEMA Handshake Inputs *)
	hiPartAvail_FromLeft			: BOOL;
	hiRdyToReceive_FromRight	: BOOL;
END_VAR
VAR_OUTPUT
	bInitialised					: BOOL;   	(*Initialisation complete flag *)
	bStopOk						: BOOL;	(* bStopOk indicates when there are no parts for processing  and FB is ok to STOP*)

	O_Drill_Spindle_On			: BOOL;	(*Drill: Turn on drill spindle.*)
	O_Drill_Fixture_Close		: BOOL;	(*Drill: Closes Fixture. Controls the valve*)

	(* Drill Zaxis control Outputs *)
	bDrill_axZ_Enable			: BOOL;	(*Drill: Z-axis: enable*)
	bDrill_axZ_Start				: BOOL;	(*Drill: Z-axis: Start motion*)
	fDrill_axZ_Velo				: REAL;	(*Drill: Z-axis: Velocity*)
	fDrill_axZ_TargetPos			: REAL;	(*Drill: Z-axis: Target position*)

	(* SMEMA Handshake Outputs *)
	hoReadyToRecieve_ToLeft	: BOOL;
	hoPartAvail_ToRight			: BOOL;

END_VAR
VAR
	bDrillHomed				: BOOL := FALSE;	(* Homing Completed Flag, only need on startup*)

	(*Timer and delay for Z axis motion block to give time for block to perform motion and clear/set flags *)
	tonMoveDelay				: TON;
	tMoveDelay				: TIME := T#1s;
	(* Drill Sequence Flags *)
	bDrill						: BOOL;
	bDrilled					: BOOL;

	bLocalReset				: BOOL := FALSE;	(*Performs local reset*)
	SFCReset 				: BOOL := FALSE;	(*Resets the execution of SFC to init once this SFCFlag is set true *)
END_VAR
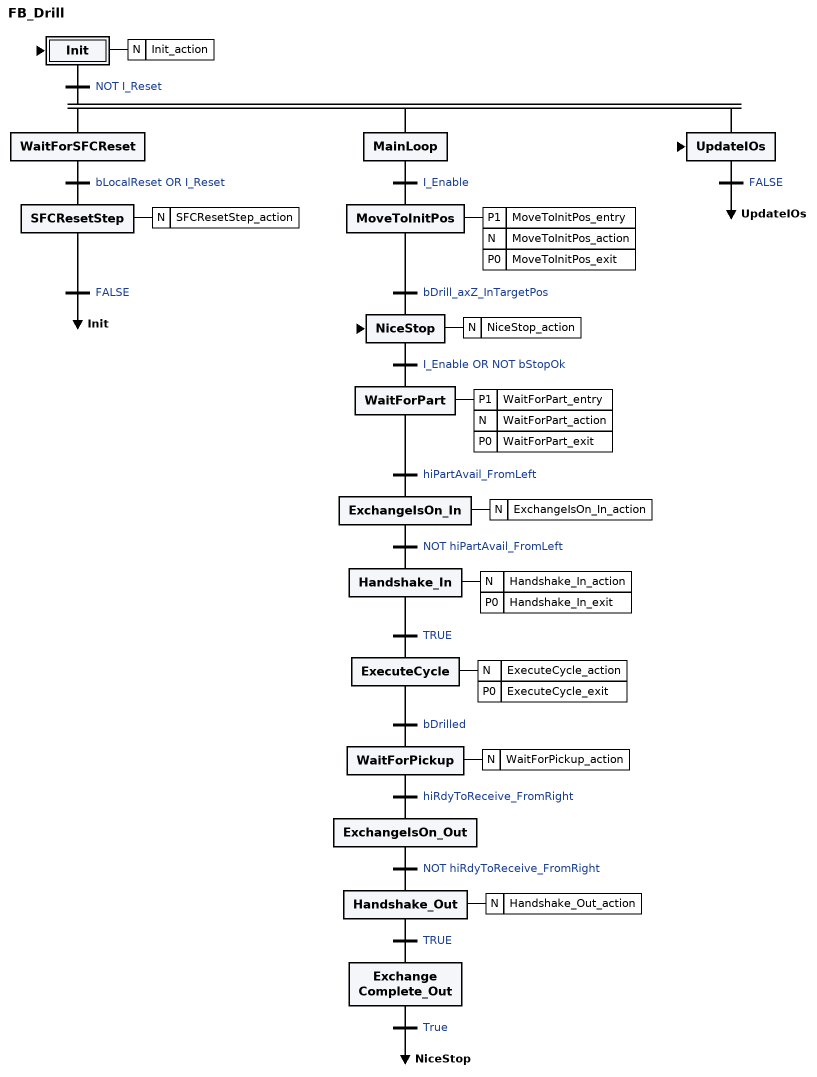
INITIAL_STEP Init:
	Init_action(N);
END_STEP
TRANSITION FROM Init TO (WaitForSFCReset, MainLoop, UpdateIOs) := NOT I_Reset;
END_TRANSITION
STEP WaitForSFCReset:
END_STEP
TRANSITION FROM WaitForSFCReset TO SFCResetStep := bLocalReset OR I_Reset;
END_TRANSITION
STEP MainLoop:
END_STEP
TRANSITION FROM MainLoop TO MoveToInitPos := I_Enable;
END_TRANSITION
STEP MoveToInitPos:
	MoveToInitPos_entry(P1);
	MoveToInitPos_action(N);
	MoveToInitPos_exit(P0);
END_STEP
TRANSITION FROM MoveToInitPos TO NiceStop := bDrill_axZ_InTargetPos;
END_TRANSITION
STEP NiceStop:
	NiceStop_action(N);
END_STEP
TRANSITION FROM NiceStop TO WaitForPart := I_Enable OR NOT bStopOk;
END_TRANSITION
STEP WaitForPart:
	WaitForPart_entry(P1);
	WaitForPart_action(N);
	WaitForPart_exit(P0);
END_STEP
TRANSITION FROM WaitForPart TO ExchangeIsOn_In := hiPartAvail_FromLeft;
END_TRANSITION
STEP ExchangeIsOn_In:
	ExchangeIsOn_In_action(N);
END_STEP
TRANSITION FROM ExchangeIsOn_In TO Handshake_In := NOT hiPartAvail_FromLeft;
END_TRANSITION
STEP Handshake_In:
	Handshake_In_action(N);
	Handshake_In_exit(P0);
END_STEP
TRANSITION FROM Handshake_In TO ExecuteCycle := TRUE;
END_TRANSITION
STEP ExecuteCycle:
	ExecuteCycle_action(N);
	ExecuteCycle_exit(P0);
END_STEP
TRANSITION FROM ExecuteCycle TO WaitForPickup := bDrilled;
END_TRANSITION
STEP WaitForPickup:
	WaitForPickup_action(N);
END_STEP
TRANSITION FROM WaitForPickup TO ExchangeIsOn_Out := hiRdyToReceive_FromRight;
END_TRANSITION
STEP ExchangeIsOn_Out:
END_STEP
TRANSITION FROM ExchangeIsOn_Out TO Handshake_Out := NOT hiRdyToReceive_FromRight;
END_TRANSITION
STEP Handshake_Out:
	Handshake_Out_action(N);
END_STEP
TRANSITION FROM Handshake_Out TO ExchangeComplete_Out := TRUE;
END_TRANSITION
STEP ExchangeComplete_Out:
END_STEP
TRANSITION FROM ExchangeComplete_Out TO NiceStop := True;
END_TRANSITION
STEP UpdateIOs:
END_STEP
TRANSITION FROM UpdateIOs TO UpdateIOs := FALSE;
END_TRANSITION
STEP SFCResetStep:
	SFCResetStep_action(N);
END_STEP
TRANSITION FROM SFCResetStep TO Init := FALSE;
END_TRANSITION

ACTION Init_action:
(* Status Flags *)
bStopOK			:= TRUE;
bInitialised 		:= FALSE;
bDrillHomed 		:= FALSE;
(* Reset Flags *)
SFCReset 		:= FALSE;
bLocalReset		:= FALSE;
(* Handshake Flags*)
hoReadyToRecieve_ToLeft	:= FALSE;
hoPartAvail_ToRight			:= FALSE;
END_ACTION

ACTION MoveToInitPos_entry:
bStopOk := FALSE;
END_ACTION

ACTION MoveToInitPos_action:
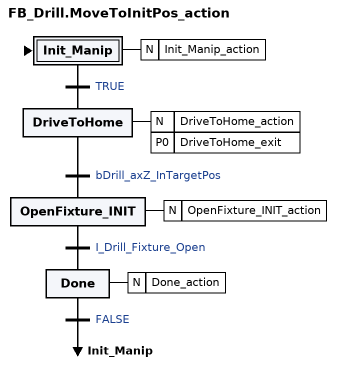
INITIAL_STEP Init_Manip:
	Init_Manip_action(N);
END_STEP
TRANSITION FROM Init_Manip TO DriveToHome := TRUE;
END_TRANSITION
STEP DriveToHome:
	DriveToHome_action(N);
	DriveToHome_exit(P0);
END_STEP
TRANSITION FROM DriveToHome TO OpenFixture_INIT := bDrill_axZ_InTargetPos;
END_TRANSITION
STEP OpenFixture_INIT:
	OpenFixture_INIT_action(N);
END_STEP
TRANSITION FROM OpenFixture_INIT TO Done := I_Drill_Fixture_Open;
END_TRANSITION
STEP Done:
	Done_action(N);
END_STEP
TRANSITION FROM Done TO Init_Manip := FALSE;
END_TRANSITION

ACTION Init_Manip_action:
bDrillHomed := FALSE;
hoReadyToRecieve_ToLeft := FALSE;
hoPartAvail_ToRight  := FALSE;
END_ACTION

ACTION DriveToHome_action:
bDrill_axZ_Enable		:= TRUE;
fDrill_axZ_TargetPos		:= -10;
fDrill_axZ_Velo			:= 5;
bDrill_axZ_Start			:= TRUE;
END_ACTION

ACTION DriveToHome_exit:
bDrill_axZ_Start := FALSE;
END_ACTION

ACTION OpenFixture_INIT_action:
O_Drill_Fixture_Close := FALSE;
END_ACTION

ACTION Done_action:
bDrillHomed := TRUE;
END_ACTION
END_ACTION

ACTION MoveToInitPos_exit:
bDrill_axZ_Start := FALSE;
bInitialised := TRUE;
END_ACTION

ACTION NiceStop_action:
(* Ok To stop if there are no parts pending from Adjacent manipulator *)
IF hiPartAvail_FromLeft THEN
	bStopOk := FALSE;
ELSE
	bStopOk := TRUE;
END_IF
END_ACTION

ACTION WaitForPart_entry:
bStopOK	:= TRUE;
END_ACTION

ACTION WaitForPart_action:
(* Set ready to recieve flag for upstream machines *)
hoReadyToRecieve_ToLeft := TRUE;
END_ACTION

ACTION WaitForPart_exit:
(* Proccessing Part, not ok to stop *)
bStopOK	:= FALSE;
END_ACTION

ACTION ExchangeIsOn_In_action:
(*Handshake Sequence *)
hoReadyToRecieve_ToLeft	:= TRUE;
END_ACTION

ACTION Handshake_In_action:
(* Handshake to indicate that part is under drill control *)
hoReadyToRecieve_ToLeft := FALSE;
END_ACTION

ACTION Handshake_In_exit:
bDrill := TRUE;
END_ACTION

ACTION ExecuteCycle_action:
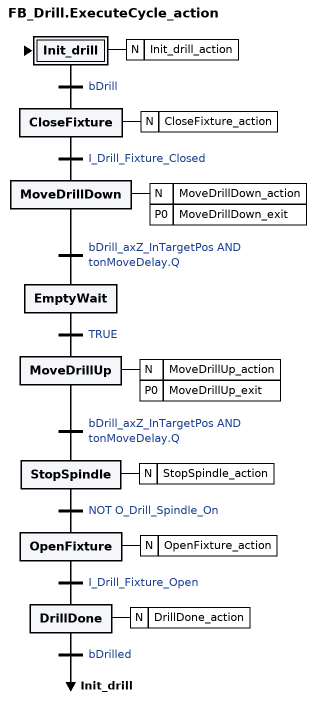
INITIAL_STEP Init_drill:
	Init_drill_action(N);
END_STEP
TRANSITION FROM Init_drill TO CloseFixture := bDrill;
END_TRANSITION
STEP CloseFixture:
	CloseFixture_action(N);
END_STEP
TRANSITION FROM CloseFixture TO MoveDrillDown := I_Drill_Fixture_Closed;
END_TRANSITION
STEP MoveDrillDown:
	MoveDrillDown_action(N);
	MoveDrillDown_exit(P0);
END_STEP
TRANSITION FROM MoveDrillDown TO EmptyWait := bDrill_axZ_InTargetPos AND tonMoveDelay.Q;
END_TRANSITION
STEP EmptyWait:
END_STEP
TRANSITION FROM EmptyWait TO MoveDrillUp := TRUE;
END_TRANSITION
STEP MoveDrillUp:
	MoveDrillUp_action(N);
	MoveDrillUp_exit(P0);
END_STEP
TRANSITION FROM MoveDrillUp TO StopSpindle := bDrill_axZ_InTargetPos AND tonMoveDelay.Q;
END_TRANSITION
STEP StopSpindle:
	StopSpindle_action(N);
END_STEP
TRANSITION FROM StopSpindle TO OpenFixture := NOT O_Drill_Spindle_On;
END_TRANSITION
STEP OpenFixture:
	OpenFixture_action(N);
END_STEP
TRANSITION FROM OpenFixture TO DrillDone := I_Drill_Fixture_Open;
END_TRANSITION
STEP DrillDone:
	DrillDone_action(N);
END_STEP
TRANSITION FROM DrillDone TO Init_drill := bDrilled;
END_TRANSITION

ACTION Init_drill_action:
O_Drill_Spindle_On	:= FALSE;
bDrill_axZ_Enable	:= FALSE;
bDrill_axZ_Start		:= FALSE;
fDrill_axZ_Velo		:= 0;
END_ACTION

ACTION CloseFixture_action:
bDrilled 					:= FALSE;
O_Drill_Fixture_Close 	:= TRUE;
END_ACTION

ACTION MoveDrillDown_action:
bDrill_axZ_Enable := TRUE;
fDrill_axZ_Velo :=10;
fDrill_axZ_TargetPos := -140;
bDrill_axZ_Start := TRUE;
tonMoveDelay(IN:=TRUE , PT:= tMoveDelay);
O_Drill_Spindle_On := TRUE;
END_ACTION

ACTION MoveDrillDown_exit:
bDrill_axZ_Start := FALSE;
tonMoveDelay(IN:=FALSE );
END_ACTION

ACTION MoveDrillUp_action:
tonMoveDelay(IN:=TRUE , PT:= tMoveDelay);
fDrill_axZ_Velo :=10;
fDrill_axZ_TargetPos := -10;
bDrill_axZ_Start := TRUE;
END_ACTION

ACTION MoveDrillUp_exit:
bDrill_axZ_Start := FALSE;
tonMoveDelay(IN:=FALSE);
END_ACTION

ACTION StopSpindle_action:
O_Drill_Spindle_On := FALSE;
END_ACTION

ACTION OpenFixture_action:
O_Drill_Fixture_Close	:= FALSE;
END_ACTION

ACTION DrillDone_action:
bDrilled := TRUE;
bDrill := FALSE;
END_ACTION
END_ACTION

ACTION ExecuteCycle_exit:
bDrilled := FALSE;
END_ACTION

ACTION WaitForPickup_action:
(* Notify downstream machine that part is avalible *)
hoPartAvail_ToRight := TRUE;
END_ACTION

ACTION Handshake_Out_action:
(* Handshake indicating part has left drill control *)
hoPartAvail_ToRight := FALSE;
END_ACTION

ACTION SFCResetStep_action:
SFCReset := TRUE;
END_ACTION
END_FUNCTION_BLOCK

(* POU Simulation/PRG_Simulator, ST *)
PROGRAM PRG_Simulator
(*This Program is simulating the real machine and mimics its behaviour.
The main task is to update the inputs for students program according the stimulus student provides as outputs.
Another task is to monitor (physical) error conditions occuring in the system and record them.
Author: Niko Siltala, niko.siltala@tut.fi, Tampere University of Technology / MEI
Date: 2016-12-12
Version: 1.0
*) 
VAR
	bBtn_EmergencyStop	: BOOL;	(*Emergency Stop button*)
	rsEmergencyClear	: RS;	(*RS - flip-flop for Emergency clear info*)
	i 	: INT;
	c 	: INT;
	fbManipLeft		: FB_Simu_Manipulator;	(*Left simulated manipulator *)
	fbManipRight	: FB_Simu_Manipulator;	(*Right simulated manipulator *)
	fbDrill			: FB_Simu_Drill;		(*Drill machine simulated*)
	arrParts_ConvIn		: ARRAY [0..10] OF ST_Part; (*Parts on input conveyour*)
	arrParts_ConvOut	: ARRAY [0..10] OF ST_Part; (*Parts on output conveyour*)
	stPart_inMLeftGripper 	: ST_Part; 	(*Data structure for the part*)
	stPart_inMRightGripper 	: ST_Part; 	(*Data structure for the part*)
	stPart_inDrillFixture 	: ST_Part; 	(*Data structure for the part*)
	bAddPartOnConvIn	: BOOL;	(*Adds new part on conveyor*)
	bClearErrors		: BOOL;	(*Clear Errors*)
	bClearSystem		: BOOL;	(*Clears system from parts *)
	RT_AddPart			: R_TRIG;
	wError_ManipL			: WORD;	(*Error bits between convIn and Manip_Left*)
	wError_Drill		: WORD; (*Error bits at drill*)
	wError_ManipR		: WORD;	(*Error bits between convIn and Manip_Left*)
	iState_IF			: ARRAY [1..5] OF UINT;	(*State variable; Exchange between 1=ConvIn->ManipL, 2=ManipL->Drill, 3=Drill->ManipR, 4=ManipR->ConvOut, 5=Drill*)
	tofPartLeavesConvOut	: TOF;	(*Off timer for out sensor*)
END_VAR
VAR CONSTANT
	bMANUAL_CONTROLS				: BOOL 	:=FALSE;(*Manual override for controls*)
	fPOS_MANIP_CONV_NO_PART_SAFE	: REAL	:= 90;	(*Manipulator on conv with NO part - Safe to move*)
	fPOS_MANIP_CONV_WITH_PART_SAFE	: REAL	:= 70;	(*Manipulator on conv with part - Safe to move*)
	fPOS_MANIP_CONV_PICK_LEVEL		: REAL	:= 120;	(*Manipulator Pick/place level on conv*)
	fPOS_MANIP_DRILL_WITH_PART_SAFE	: REAL	:= 53;	(*Manipulator coming to drill with part - Safe to move*)
	fPOS_MANIP_DRILL_NO_PART_SAFE	: REAL	:= 46;	(*Manipulator coming to drill with NO part - Safe to move*)
	fPOS_MANIP_DRILL_PICK_LEVEL		: REAL	:= 74;	(*Manipulator Pick/place level on Drill*)
	fPOS_MANIP_PICK_TOLERANCE		: REAL	:= 30;	(*Manipulator Pick level tolerance from the part (=fingers length)*)
	fPART_HEIGH						: REAL	:= 50;	(*Part height*)
	fPART_PICK_TOLERANCE			: REAL	:= 10;	(*Part pick & place (negative) tolerance from Levels.*)
	fPART_HOLE_DEPTH_REQ			: REAL	:= 40;	(*Part required Hole depth*)
	fPART_HOLE_DEPTH_MAX			: REAL	:= 45;	(*Max Hole depth*)
	fPOS_DRILL_BIT_TOUCHES			: REAL	:= 100;	(*Drill touches the part*)
	iDRILL_SPINDLE_MIN_FOR_DRILLING	: INT	:= 400;	(*Minimum spindle speed for drilling*)
END_VAR
(*Handle counter*)
c:= c+1;
IF c> 10 THEN
	c:= 0;
END_IF;

(*Simulate emergency stop circuitry*)
rsEmergencyClear(
	SET:= I_Btn_Reset,
	RESET1:= bBtn_EmergencyStop,
	Q1=> I_EmergencyClear);

(*Adds new parts on input conveyour*)
RT_AddPart(CLK:=bAddPartOnConvIn , Q=> );
IF RT_AddPart.Q AND NOT arrParts_ConvIn[5].bExists THEN
	arrParts_ConvIn[5].bExists := TRUE;
END_IF;

(*Input Conveyour Simulation*)
IF O_ConvIn_MotON THEN
	IF (c MOD 5) = 0 THEN
		(*Move parts forward*)
		F_MovePartForward(arrParts_ConvIn);
	END_IF;
END_IF;
(*Part in pick postition*)
I_ConvIn_PartPresent := arrParts_ConvIn[0].bExists;

(*Output Conveyour Simulation*)
IF O_ConvOut_MotON THEN
	IF (c MOD 5) = 0 THEN
		(*Move parts forward*)
		F_MovePartForward(arrParts_ConvOut);
	END_IF;
END_IF;
(*Part in end postition*)
I_ConvOut_PartPresent := arrParts_ConvOut[0].bExists;
tofPartLeavesConvOut(
	IN:=arrParts_ConvOut[0].bExists ,
	PT:= T#1s,
	Q=>I_ConvOut_PartPresent );
IF arrParts_ConvOut[0].bExists THEN
	(*Clear part at end of output conveyour*)
	arrParts_ConvOut[0].bExists := FALSE;
	arrParts_ConvOut[0].bHasHole := FALSE;
END_IF;


IF bMANUAL_CONTROLS THEN
	(*Left manipulator*)
	fbManipLeft(
		bEnable:= ,
		bLift_Start:= ,
		fLift_Velo:= ,
		fLift_TargetPos:= ,
		bBeam_Left:= ,
		bBeam_Right:= ,
		bGripper_Close:= ,
		stPart_inGripper:= stPart_inMLeftGripper,
		bGripperIsOpen=> I_ManiL_Gripper_Open,
		bLift_InTarget=> bManiL_axZ_InTargetPos,
		fLift_CurrentPos=> fManiL_axZ_CurrPos,
		bLimit_Top=> I_ManiL_Limit_Up,
		bLimit_Bottom=> I_ManiL_Limit_Dn,
		bHome_Sensor=> I_ManiL_Limit_Home,
		bBeamAtRight=> I_ManiL_Turned_Right,
		bBeamAtLeft=> I_ManiL_Turned_Left);
	
	(*Right manipulator*)
	fbManipRight(
		bEnable:= ,
		bLift_Start:= ,
		fLift_Velo:= , 
		fLift_TargetPos:= , 
		bBeam_Left:= ,
		bBeam_Right:= ,
		bGripper_Close:= , 
		stPart_inGripper:= stPart_inMRightGripper,
		bGripperIsOpen=> I_ManiR_Gripper_Open,
		bLift_InTarget=> bManiR_axZ_InTargetPos,
		fLift_CurrentPos=> fManiR_axZ_CurrPos,
		bLimit_Top=> I_ManiR_Limit_Up,
		bLimit_Bottom=> I_ManiR_Limit_Dn,
		bHome_Sensor=> I_ManiR_Limit_Home,
		bBeamAtRight=> I_ManiR_Turned_Right,
		bBeamAtLeft=> I_ManiR_Turned_Left);
	
	(*Call drill machine*)
	fbDrill(
		bEnable:= ,
		bLift_Start:= ,
		fLift_Velo:= ,
		fLift_TargetPos:= , 
		bDrillOn:= , 
		bFixture_Close:= , 
		stPart_inFixture:= stPart_inDrillFixture,
		bLift_InTarget=> bDrill_axZ_InTargetPos,
		fLift_CurrentPos=> fDrill_axZ_CurrPos,
		bLimit_Top=> I_Drill_Limit_Up,
		bLimit_Bottom=> I_Drill_Limit_Dn,
		bHome_Sensor=> I_Drill_Limit_Home,
		bFixture_Open=> I_Drill_Fixture_Open,
		bFixture_Closed=> I_Drill_Fixture_Closed);

ELSE
	(*Left manipulator*)
	fbManipLeft(
		bEnable:= bManiL_axZ_Enable,
		bLift_Start:= bManiL_axZ_Start,
		fLift_Velo:= fManiL_axZ_Velo,
		fLift_TargetPos:= fManiL_axZ_TargetPos,
		bBeam_Left:= O_ManiL_Turn_Left,
		bBeam_Right:= O_ManiL_Turn_Right,
		bGripper_Close:= O_ManiL_Gripper_Close,
		stPart_inGripper:= stPart_inMLeftGripper,
		bGripperIsOpen=> I_ManiL_Gripper_Open,
		bLift_InTarget=> bManiL_axZ_InTargetPos,
		fLift_CurrentPos=> fManiL_axZ_CurrPos,
		bLimit_Top=> I_ManiL_Limit_Up,
		bLimit_Bottom=> I_ManiL_Limit_Dn,
		bHome_Sensor=> I_ManiL_Limit_Home,
		bBeamAtRight=> I_ManiL_Turned_Right,
		bBeamAtLeft=> I_ManiL_Turned_Left);

	(*Right manipulator*)
	fbManipRight(
		bEnable:= bManiR_axZ_Enable,
		bLift_Start:= bManiR_axZ_Start,
		fLift_Velo:= fManiR_axZ_Velo,
		fLift_TargetPos:= fManiR_axZ_TargetPos,
		bBeam_Left:= O_ManiR_Turn_Left,
		bBeam_Right:= O_ManiR_Turn_Right,
		bGripper_Close:= O_ManiR_Gripper_Close,
		stPart_inGripper:= stPart_inMRightGripper,
		stPart_inGripper:= stPart_inMRightGripper,
		bGripperIsOpen=> I_ManiR_Gripper_Open,
		bLift_InTarget=> bManiR_axZ_InTargetPos,
		fLift_CurrentPos=> fManiR_axZ_CurrPos,
		bLimit_Top=> I_ManiR_Limit_Up,
		bLimit_Bottom=> I_ManiR_Limit_Dn,
		bHome_Sensor=> I_ManiR_Limit_Home,
		bBeamAtRight=> I_ManiR_Turned_Right,
		bBeamAtLeft=> I_ManiR_Turned_Left);

	(*Call drill machine*)
	fbDrill(
		bEnable:= bDrill_axZ_Enable,
		bLift_Start:= bDrill_axZ_Start,
		fLift_Velo:= fDrill_axZ_Velo,
		fLift_TargetPos:= fDrill_axZ_TargetPos,
		bDrillOn:= O_Drill_Spindle_On,
		bFixture_Close:= O_Drill_Fixture_Close,
		stPart_inFixture:= stPart_inDrillFixture,
		bLift_InTarget=> bDrill_axZ_InTargetPos,
		fLift_CurrentPos=> fDrill_axZ_CurrPos,
		bLimit_Top=> I_Drill_Limit_Up,
		bLimit_Bottom=> I_Drill_Limit_Dn,
		bHome_Sensor=> I_Drill_Limit_Home,
		bFixture_Open=> I_Drill_Fixture_Open,
		bFixture_Closed=> I_Drill_Fixture_Closed);
END_IF;


(*Make part exchange and check error conditions between ConvIn and ManipLeft*)
ErrorCheck_ManipLeft_ConvIn;
(*Make part exchange and check error conditions between ManipLeft and Drill*)
ErrorCheck_ManipLeft_Drill;
(*Make drilling and check error conditions at Drilling*)
ErrorCheck_Drill;
(*Make part exchange and check error conditions between ManipRight and Drill*)
ErrorCheck_ManipRight_Drill;
(*Make part exchange and check error conditions between ManipRight and ConvOut*)
ErrorCheck_ManipRight_ConvOut;
(*Collisions between devices*)
ErrorCheck_Collisions;


(*drops part from Manipulator Left*)
IF stPart_inMLeftGripper.bExists AND fbManipLeft.bGripperIsOpen THEN
	stPart_inMLeftGripper.bExists := FALSE;
END_IF;
(*drops part from Manipulator Right*)
IF stPart_inMRightGripper.bExists AND fbManipRight.bGripperIsOpen THEN
	stPart_inMRightGripper.bExists := FALSE;
END_IF;



(*Clear active errors*)
IF bClearErrors THEN
	wError_ManipL := 0;
	wError_Drill := 0;
	wError_ManipR := 0;
END_IF;

(*Remove parts from entire system*)
IF bClearSystem THEN
	(*Clear input & output conveyour from parts*)
	FOR i:= 0 TO 10 DO
		arrParts_ConvIn[i].bExists := FALSE;
		arrParts_ConvOut[i].bExists := FALSE;
	END_FOR;
	(*Clear Manipulators and drill from parts*)
	stPart_inMLeftGripper.bExists := FALSE;
	stPart_inDrillFixture.bExists := FALSE;
	stPart_inMRightGripper.bExists := FALSE;
END_IF;
END_PROGRAM
ACTION ErrorCheck_Collisions:
(*ManipL and Conveyor collision*)
IF (fbManipLeft.fPos_Y > 140) AND (fbManipLeft.fPos_angle < 50) THEN
	wError_ManipL.7 := TRUE;	(*collision with conveyor*)
END_IF;

(*ManipL and Drill collision*)
IF ((fbDrill.fPos_Y + 16) > fbManipLeft.fPos_Y) AND fbManipLeft.fPos_angle > 150 THEN
	wError_ManipL.1 := TRUE;
	wError_Drill.0 := TRUE;
END_IF;

(*ManipR and Drill collision*)
IF ((fbDrill.fPos_Y + 10) > fbManipRight.fPos_Y) AND fbManipRight.fPos_angle < 40 THEN	(* was +16 and <50 *)
	wError_ManipR.1 := TRUE;
	wError_Drill.1 := TRUE;
END_IF;

(*ManipR and Conveyor collision*)
IF (fbManipRight.fPos_Y > 140) AND (fbManipRight.fPos_angle > 150) THEN
	wError_ManipR.7 := TRUE;	(*collision with conveyor*)
END_IF;

(*ManipL and ManipR collision*)
IF (fbManipLeft.fPos_angle > 130) AND (fbManipRight.fPos_angle < 50) AND
  (ABS(fbManipRight.fPos_Y - fbManipLeft.fPos_Y) < 60) THEN
	wError_ManipL.9 := TRUE;	(*collision sidewise with ManipulatorRight*)
	wError_ManipR.9 := TRUE;	(*collision sidewise with ManipulatorLeft*)
END_IF;
END_ACTION
ACTION ErrorCheck_Drill:
(*State model for Drilling.
Includes all associated error conditions and judgements *)

(*Drilling cycle has been initiated, but part is removed somewhere between.*)
IF (iState_IF[5] > 0) AND NOT stPart_inDrillFixture.bExists THEN
	iState_IF[5] := 0;
END_IF;

(*Drilled too long*)
IF stPart_inDrillFixture.bExists AND
  (fbDrill.fPos_Y > (fPOS_DRILL_BIT_TOUCHES + fPART_HOLE_DEPTH_MAX)) THEN
	wError_Drill.2 := TRUE;	(*collision with part and Drill*)
END_IF;


CASE iState_IF[5] OF
0: (* IDLE *)
	IF fbDrill.fPos_Y > ( fPOS_DRILL_BIT_TOUCHES - fPART_HEIGH ) THEN
		iState_IF[5] := 1;
	END_IF;

1: (* Approaches with Drill *)
	IF  fbDrill.fPos_Y >= fPOS_DRILL_BIT_TOUCHES THEN
		iState_IF[5] := 2;
	END_IF;

2: (* Drilling *)
	IF fbDrill.fPos_Y >= (fPOS_DRILL_BIT_TOUCHES + fPART_HOLE_DEPTH_REQ ) THEN
		iState_IF[5] := 3;
	END_IF;
	IF stPart_inDrillFixture.bExists AND NOT fbDrill.bFixture_Closed THEN
		wError_Drill.7 := TRUE;	(*Drilling without closed fixture*)
	END_IF;
	IF stPart_inDrillFixture.bExists AND fbDrill.iRPMCurrent < iDRILL_SPINDLE_MIN_FOR_DRILLING THEN
		wError_Drill.2 := TRUE;	(*collision with part and Drill*)
		wError_Drill.6 := TRUE;	(*Drilling without sufficient spindle RPM*)
	END_IF;

3: (* Drilled *)
	stPart_inDrillFixture.bHasHole := TRUE;
	IF fbDrill.fPos_Y < fPOS_DRILL_BIT_TOUCHES THEN
		iState_IF[5] := 4;
	END_IF;

4: (* moved up from part *)
	stPart_inDrillFixture.bHasHole := TRUE;
	IF fbDrill.fPos_Y < 30 THEN
		iState_IF[5] := 5;
	END_IF;

5: (* moved to wait area *)
	iState_IF[5] := 0;

ELSE
	iState_IF[5] := 0;
END_CASE;
END_ACTION
ACTION ErrorCheck_ManipLeft_ConvIn:
(*State model for exchanging part from ConveyorIn to ManipLeft.
Includes all associated error conditions and judgements *)

CASE iState_IF[1] OF
0: (* IDLE *)
	IF arrParts_ConvIn[0].bExists AND NOT stPart_inMLeftGripper.bExists THEN
		iState_IF[1] := 1;
	END_IF;

1: (* waitMoveAbove *)
	IF fbManipLeft.bBeamAtLeft AND fbManipLeft.fPos_Y < fPOS_MANIP_CONV_NO_PART_SAFE THEN
		iState_IF[1] := 2;
	END_IF;
	IF fbManipLeft.fPos_angle < 30 AND fbManipLeft.fPos_Y > fPOS_MANIP_CONV_NO_PART_SAFE THEN
		wError_ManipL.0 := TRUE;
	END_IF;

2: (* ManipulatorLeft is above *)
	IF fbManipLeft.bBeamAtLeft AND fbManipLeft.fPos_Y >= fPOS_MANIP_CONV_NO_PART_SAFE THEN
		iState_IF[1] := 3;
	END_IF;
	IF NOT fbManipLeft.bBeamAtLeft AND fbManipLeft.fPos_angle < 30 AND fbManipLeft.fPos_Y > fPOS_MANIP_CONV_NO_PART_SAFE THEN
		wError_ManipL.0 := TRUE;
	END_IF;

3: (* Approaches from above *)
	IF fbManipLeft.bBeamAtLeft AND fbManipLeft.bGripperIsOpen AND
	  fbManipLeft.fPos_Y >= (fPOS_MANIP_CONV_PICK_LEVEL - 2*fPART_PICK_TOLERANCE) THEN
		iState_IF[1] := 4;
	ELSIF fbManipLeft.fPos_Y < fPOS_MANIP_CONV_NO_PART_SAFE THEN
		iState_IF[1] := 0;
	END_IF;
	IF NOT fbManipLeft.bBeamAtLeft THEN
		wError_ManipL.0 := TRUE;
	END_IF;
	IF NOT fbManipLeft.bGripperIsOpen THEN
		wError_ManipL.5 := TRUE;
	END_IF;

4: (* Over part *)
	IF fbManipLeft.bBeamAtLeft AND fbManipLeft.fPos_Y >= (fPOS_MANIP_CONV_PICK_LEVEL - fPART_PICK_TOLERANCE) AND
	fbManipLeft.fPos_Y <= fPOS_MANIP_CONV_PICK_LEVEL AND fbManipLeft.bGripperClosed THEN
		(*Grasping occurs*)
		iState_IF[1] := 5;
		(*TODO: Add part grasp height compensation*)
	ELSIF fbManipLeft.fPos_Y < fPOS_MANIP_CONV_NO_PART_SAFE THEN
		iState_IF[1] := 0;
	END_IF;
	IF NOT fbManipLeft.bBeamAtLeft THEN
		wError_ManipL.0 := TRUE;
	END_IF;
	IF fbManipLeft.fPos_Y > fPOS_MANIP_CONV_PICK_LEVEL THEN
		wError_ManipL.2 := TRUE;
	END_IF;

5: (* part grasped *)
	stPart_inMLeftGripper.bExists := TRUE;
	IF fbManipLeft.bBeamAtLeft AND fbManipLeft.fPos_Y < fPOS_MANIP_CONV_WITH_PART_SAFE THEN
		iState_IF[1] := 6;
	END_IF;
	IF NOT fbManipLeft.bBeamAtLeft AND fbManipLeft.fPos_Y > fPOS_MANIP_CONV_NO_PART_SAFE THEN
		wError_ManipL.3 := TRUE;
	END_IF;

6: (* moved up with part *)
	IF fbManipLeft.fPos_Y < fPOS_MANIP_CONV_WITH_PART_SAFE THEN
		iState_IF[1] := 7;
	END_IF;

7: (* moved up with part *)
	arrParts_ConvIn[0].bExists := FALSE;
	iState_IF[1] := 0;

ELSE
	iState_IF[1] := 0;
END_CASE;
END_ACTION
ACTION ErrorCheck_ManipLeft_Drill:
(*State model for exchanging part from ManipLeft to Drill.
Includes all associated error conditions and judgements *)

(*Dropping part from gripper too soon*)
IF (iState_IF[2] > 0) AND (iState_IF[2] <= 3) AND NOT fbManipLeft.bGripperClosed AND stPart_inMLeftGripper.bExists THEN
	wError_ManipL.6 := TRUE;
	iState_IF[2] := 0;
END_IF;

(*Collision with parts*)
IF stPart_inMLeftGripper.bExists AND stPart_inDrillFixture.bExists AND fbManipLeft.bBeamAtRight AND
  fbManipLeft.fPos_Y > (fPOS_MANIP_DRILL_PICK_LEVEL - 2* fPART_HEIGH) THEN
	wError_Drill.3 := TRUE;
END_IF;

(*Part exchange sequence*)
CASE iState_IF[2] OF
0: (* IDLE *)
	IF stPart_inMLeftGripper.bExists AND fbManipLeft.bGripperClosed THEN
		iState_IF[2] := 1;
	END_IF;

1: (* waitMoveAbove *)
	IF fbManipLeft.bBeamAtRight AND fbManipLeft.fPos_Y < fPOS_MANIP_DRILL_WITH_PART_SAFE THEN
		iState_IF[2] := 2;
	END_IF;
	IF fbManipLeft.fPos_angle > 150 AND fbManipLeft.fPos_Y > fPOS_MANIP_DRILL_WITH_PART_SAFE THEN
		wError_ManipL.1 := TRUE;
	END_IF;

2: (* ManipulatorLeft is above release point*)
	IF fbManipLeft.bBeamAtRight AND fbManipLeft.fPos_Y >= fPOS_MANIP_DRILL_WITH_PART_SAFE THEN
		iState_IF[2] := 3;
	END_IF;
	IF NOT fbManipLeft.bBeamAtRight AND (fbManipLeft.fPos_angle > 150) AND
	  (fbManipLeft.fPos_Y > fPOS_MANIP_DRILL_WITH_PART_SAFE) THEN
		wError_ManipL.1 := TRUE;
	END_IF;

3: (* Approaches from above *)
	IF fbManipLeft.bBeamAtRight AND fbManipLeft.bGripperClosed AND
	  (fbManipLeft.fPos_Y >= (fPOS_MANIP_DRILL_PICK_LEVEL - fPART_PICK_TOLERANCE)) THEN
		iState_IF[2] := 4;
	ELSIF fbManipLeft.fPos_Y < fPOS_MANIP_DRILL_WITH_PART_SAFE THEN
		iState_IF[2] := 0;
	END_IF;
	IF NOT fbManipLeft.bBeamAtRight AND fbManipLeft.fPos_Y > fPOS_MANIP_DRILL_WITH_PART_SAFE THEN
		wError_ManipL.1 := TRUE;
	END_IF;

4: (* At release point *)
	(*Errors*)
	IF stPart_inDrillFixture.bExists THEN
		wError_ManipL.2 := TRUE;
		wError_Drill.3 := TRUE;
	END_IF;
	(*State trensition*)
	IF fbManipLeft.bBeamAtRight AND (fbManipLeft.fPos_Y >= (fPOS_MANIP_DRILL_PICK_LEVEL - fPART_PICK_TOLERANCE)) AND
	fbManipLeft.fPos_Y <= fPOS_MANIP_DRILL_PICK_LEVEL AND fbManipLeft.bGripperIsOpen THEN
		(*Release occurs*)
		iState_IF[2] := 5;
		(*Copy part to Drill Fixture*)
		F_CopyPart(stPart_inMLeftGripper, stPart_inDrillFixture);
		stPart_inMLeftGripper.bExists := FALSE;
	ELSIF fbManipLeft.fPos_Y < fPOS_MANIP_DRILL_WITH_PART_SAFE THEN
		iState_IF[2] := 0;
	END_IF;
	IF NOT fbManipLeft.bBeamAtRight AND fbManipLeft.fPos_Y > fPOS_MANIP_DRILL_WITH_PART_SAFE THEN
		wError_ManipL.1 := TRUE;
	END_IF;
	IF fbManipLeft.fPos_Y > fPOS_MANIP_DRILL_PICK_LEVEL THEN
		wError_ManipL.2 := TRUE;
	END_IF;
	IF fbDrill.bFixture_Closed THEN
		wError_Drill.4 := TRUE;	(*Fixture closed when inserting part*)
	END_IF;

5: (* Release part *)
	IF fbManipLeft.bBeamAtRight AND fbManipLeft.fPos_Y <= fPOS_MANIP_DRILL_NO_PART_SAFE THEN
		iState_IF[2] := 6;
	ELSIF fbManipLeft.bBeamAtLeft AND fbManipLeft.fPos_Y <= fPOS_MANIP_CONV_NO_PART_SAFE THEN
		(* Errornous leave condition*)
		iState_IF[2] := 0;
	END_IF;
	IF NOT fbManipLeft.bBeamAtRight AND fbManipLeft.fPos_Y > fPOS_MANIP_DRILL_NO_PART_SAFE THEN
		wError_ManipL.1 := TRUE;
		wError_ManipL.3 := TRUE;
	END_IF;
	IF NOT fbManipLeft.bGripperIsOpen THEN
		wError_ManipR.10 := TRUE;	(*re-grasping released part*)
	END_IF;

6: (* moved up *)
	IF fbManipLeft.fPos_Y <= fPOS_MANIP_DRILL_NO_PART_SAFE THEN
		iState_IF[2] := 7;
	END_IF;
	iState_IF[2] := 0;

7: (* Can move away *)
	iState_IF[2] := 0;

ELSE
	iState_IF[2] := 0;
END_CASE;
END_ACTION
ACTION ErrorCheck_ManipRight_ConvOut:
(*State model for exchanging part from ManipRight to Conveyor.
Includes all associated error conditions and judgements *)

(*Dropping part from gripper too soon*)
IF (iState_IF[4] > 0) AND (iState_IF[4] <= 3) AND NOT fbManipRight.bGripperClosed AND stPart_inMRightGripper.bExists THEN
	wError_ManipR.6 := TRUE;
	iState_IF[4] := 0;
END_IF;

(*Collision with parts*)
IF stPart_inMRightGripper.bExists AND arrParts_ConvOut[5].bExists AND fbManipRight.fPos_angle > 150 AND
  fbManipRight.fPos_Y > (fPOS_MANIP_CONV_PICK_LEVEL - fPART_HEIGH) THEN
	wError_ManipR.8 := TRUE;
END_IF;

(*Part exchange sequence*)
CASE iState_IF[4] OF
0: (* IDLE *)
	IF stPart_inMRightGripper.bExists AND fbManipRight.bGripperClosed THEN
		iState_IF[4] := 1;
	END_IF;

1: (* waitMoveAbove *)
	IF fbManipRight.bBeamAtRight AND fbManipRight.fPos_Y <= fPOS_MANIP_CONV_WITH_PART_SAFE THEN
		iState_IF[4] := 2;
	END_IF;
	IF fbManipRight.fPos_angle > 150 AND fbManipRight.fPos_Y > fPOS_MANIP_CONV_WITH_PART_SAFE THEN
		wError_ManipR.0 := TRUE;
	END_IF;

2: (* ManipulatorRight is above release point*)
	IF fbManipRight.bBeamAtRight AND fbManipRight.fPos_Y >= fPOS_MANIP_CONV_WITH_PART_SAFE THEN
		iState_IF[4] := 3;
	END_IF;
	IF NOT fbManipRight.bBeamAtRight AND (fbManipRight.fPos_angle > 150) AND
	  (fbManipRight.fPos_Y > fPOS_MANIP_CONV_WITH_PART_SAFE) THEN
		wError_ManipR.0 := TRUE;
	END_IF;

3: (* Approaches from above *)
	IF fbManipRight.bBeamAtRight AND fbManipRight.bGripperClosed AND
	  (fbManipRight.fPos_Y >= (fPOS_MANIP_CONV_PICK_LEVEL - fPART_PICK_TOLERANCE)) THEN
		iState_IF[4] := 4;
	ELSIF fbManipRight.fPos_Y < fPOS_MANIP_CONV_WITH_PART_SAFE THEN
		iState_IF[4] := 0;
	END_IF;
	IF NOT fbManipRight.bBeamAtRight AND fbManipRight.fPos_Y > fPOS_MANIP_CONV_WITH_PART_SAFE THEN
		wError_ManipR.0 := TRUE;
	END_IF;

4: (* At release point *)
	(*Errors*)
	IF arrParts_ConvOut[5].bExists THEN
		wError_ManipR.2 := TRUE;
	END_IF;
	(*State trensition*)
	IF fbManipRight.bBeamAtRight AND (fbManipRight.fPos_Y >= (fPOS_MANIP_CONV_PICK_LEVEL - fPART_PICK_TOLERANCE)) AND
	fbManipRight.fPos_Y <= fPOS_MANIP_CONV_PICK_LEVEL AND fbManipRight.bGripperIsOpen THEN
		(*Release occurs*)
		iState_IF[4] := 5;
		(*Copy part to Conveyour Out*)
		F_CopyPart(stPart_inMRightGripper, arrParts_ConvOut[5]);
		(*TODO: Add part grasp height compensation*)
	ELSIF fbManipRight.fPos_Y < fPOS_MANIP_CONV_WITH_PART_SAFE THEN
		iState_IF[4] := 0;
	END_IF;
	IF NOT fbManipRight.bBeamAtRight AND fbManipRight.fPos_Y > fPOS_MANIP_CONV_WITH_PART_SAFE THEN
		wError_ManipR.1 := TRUE;
	END_IF;
	IF fbManipRight.fPos_Y > fPOS_MANIP_CONV_PICK_LEVEL THEN
		wError_ManipR.2 := TRUE;
	END_IF;

5: (* Release part *)
	stPart_inMRightGripper.bExists := FALSE;
	IF fbManipRight.bBeamAtRight AND fbManipRight.fPos_Y <= fPOS_MANIP_CONV_NO_PART_SAFE AND
	   fbManipRight.bGripperIsOpen THEN
		iState_IF[4] := 6;
	END_IF;
	IF NOT fbManipRight.bBeamAtRight AND fbManipRight.fPos_Y > fPOS_MANIP_CONV_NO_PART_SAFE THEN
		wError_ManipR.1 := TRUE;
		wError_ManipR.3 := TRUE;
	END_IF;
	IF NOT fbManipRight.bGripperIsOpen THEN
		wError_ManipR.10 := TRUE;	(*re-grasping released part*)
	END_IF;

6: (* moved up *)
	iState_IF[4] := 0;

ELSE
	iState_IF[4] := 0;
END_CASE;
END_ACTION
ACTION ErrorCheck_ManipRight_Drill:
(*State model for exchanging part from Drive to ManipRight.
Includes all associated error conditions and judgements *)

CASE iState_IF[3] OF
0: (* IDLE *)
	IF stPart_inDrillFixture.bExists AND NOT stPart_inMRightGripper.bExists THEN
		iState_IF[3] := 1;
	END_IF;

1: (* waitMoveAbove *)
	IF fbManipRight.bBeamAtLeft AND fbManipRight.fPos_Y <= fPOS_MANIP_DRILL_NO_PART_SAFE THEN
		iState_IF[3] := 2;
	END_IF;
	IF fbManipRight.fPos_angle < 30 AND fbManipRight.fPos_Y > fPOS_MANIP_DRILL_NO_PART_SAFE THEN
		wError_ManipR.1 := TRUE;
	END_IF;

2: (* ManipulatorLeft is above *)
	IF fbManipRight.bBeamAtLeft AND fbManipRight.fPos_Y >= fPOS_MANIP_DRILL_NO_PART_SAFE THEN
		iState_IF[3] := 3;
	END_IF;
	IF NOT fbManipRight.bBeamAtLeft AND fbManipRight.fPos_angle > 30 AND fbManipRight.fPos_Y > fPOS_MANIP_DRILL_NO_PART_SAFE THEN
		wError_ManipR.1 := TRUE;
	END_IF;

3: (* Approaches from above *)
	IF fbManipRight.bBeamAtLeft AND fbManipRight.bGripperIsOpen AND
	  fbManipRight.fPos_Y >= (fPOS_MANIP_DRILL_PICK_LEVEL - fPART_PICK_TOLERANCE) THEN
		iState_IF[3] := 4;
	ELSIF fbManipRight.fPos_Y < fPOS_MANIP_DRILL_NO_PART_SAFE THEN
		iState_IF[3] := 0;
	END_IF;
	IF NOT fbManipRight.bBeamAtLeft THEN
		wError_ManipR.1 := TRUE;
	END_IF;
	IF NOT fbManipRight.bGripperIsOpen THEN
		wError_ManipR.5 := TRUE;
	END_IF;

4: (* Over part *)
	IF fbManipRight.bBeamAtLeft AND fbManipRight.fPos_Y >= (fPOS_MANIP_DRILL_PICK_LEVEL - fPART_PICK_TOLERANCE) AND
	fbManipRight.fPos_Y <= fPOS_MANIP_DRILL_PICK_LEVEL AND fbManipRight.bGripperClosed THEN
		(*Grasping occurs*)
		iState_IF[3] := 5;
		(*Copy part from Drill Fixture*)
		F_CopyPart(stPart_inDrillFixture, stPart_inMRightGripper);
		(*TODO: Add part grasp height compensation*)
		stPart_inDrillFixture.bExists := FALSE;
		stPart_inDrillFixture.bHasHole := FALSE;
	ELSIF fbManipRight.fPos_Y < fPOS_MANIP_DRILL_NO_PART_SAFE THEN
		iState_IF[3] := 0;
	END_IF;
	IF NOT fbManipRight.bBeamAtLeft THEN
		wError_ManipR.1 := TRUE;
	END_IF;
	IF fbManipRight.fPos_Y > fPOS_MANIP_DRILL_PICK_LEVEL THEN
		wError_ManipR.2 := TRUE;
	END_IF;

5: (* part grasped *)
	IF fbManipRight.bBeamAtLeft AND fbManipRight.fPos_Y < (fPOS_MANIP_DRILL_PICK_LEVEL - fPART_PICK_TOLERANCE) THEN
		iState_IF[3] := 6;
	END_IF;
	IF NOT fbManipRight.bBeamAtLeft AND fbManipRight.fPos_Y > fPOS_MANIP_DRILL_WITH_PART_SAFE THEN
		wError_ManipR.3 := TRUE;
	END_IF;

6: (* leaving with part *)
	IF fbManipRight.bBeamAtLeft AND fbManipRight.fPos_Y <= fPOS_MANIP_DRILL_WITH_PART_SAFE THEN
		iState_IF[3] := 7;
	END_IF;
	IF NOT fbManipRight.bBeamAtLeft AND fbManipRight.fPos_Y > fPOS_MANIP_DRILL_WITH_PART_SAFE THEN
		wError_ManipR.3 := TRUE; 	(*Fixture closed while leaving with part*)
	END_IF;
	IF fbDrill.bFixture_Closed THEN
		wError_Drill.5 := TRUE;	(*Fixture closed while leaving with part*)
	END_IF;

7: (* moved up with part *)
	iState_IF[3] := 0;

ELSE
	iState_IF[3] := 0;
END_CASE;
END_ACTION

(* POU Simulation/FB_Simu_Manipulator, ST *)
FUNCTION_BLOCK FB_Simu_Manipulator
(*Simulation model for the behaviour of the Manipulator.
Author: Niko Siltala, niko.siltala@tut.fi, Tampere University of Technology / MEI
Date: 2016-12-12
Version: 1.0
*)
VAR_INPUT
	bEnable			: BOOL := TRUE;	(*Enable manipulator*)
	bLift_Start		: BOOL;	(*Triggers and starts the lift movement at rising edge*)
	fLift_Velo		: REAL := 10;	(*Velocity*)
	fLift_TargetPos	: REAL;	(*Target position*)
	bBeam_Left		: BOOL;	(*Turn beam at left*)
	bBeam_Right		: BOOL;	(*Turn beam at right*)
	bGripper_Close	: BOOL; (*Close Gripper*)
END_VAR
VAR_OUTPUT
	bGripperIsOpen	: BOOL;	(*Gripper is open*)
	bLift_InTarget	: BOOL;	(*Lift has reached the target*)
	fLift_CurrentPos	: REAL;	(*Current position of the lift*)
	bLimit_Top		: BOOL;	(*Height position at top limit*)
	bLimit_Bottom	: BOOL;	(*Height position at bottom limit*)
	bHome_Sensor	: BOOL;	(*Height position at home limit*)
	bBeamAtRight	: BOOL;	(*Beam turned into right limit*)
	bBeamAtLeft		: BOOL;	(*Beam turned into left limit*)
END_VAR
VAR_IN_OUT
	stPart_inGripper : ST_Part; 	(*Data structure for the part*)
END_VAR
VAR
	fPos_angle	: REAL := 70;	(*Angle of beam [deg]*)
	fPos_height	: REAL;	(* Manipulators height position*)
	fPos_X		: REAL;	(* Manipulator's X position*)
	fPos_Y		: REAL;	(* Manipulator's Y position*)
	fBasePos_Y 	: REAL; (*Position of manipulator base*)
	iState_Lift		: UINT;	(*State of beam model*)
	fPos_Beam_L	: REAL;	(*Beam position left end*)
	fPos_Beam_R	: REAL;	(*Beam position right end*)
	bGripperClosed	: BOOL; (*Gripper is closed*)
	fPosFingerDiff 	: REAL;	(*Right finger position. 0 poistion when grasping.*)
	bInitDone		: BOOL;		(*Initialisation done for simulated machine*)
END_VAR
VAR CONSTANT
	iBEAM_LENGTH	: USINT := 120;	(*length of the beam*)
	fPOS_MAX_DOWN	: REAL	:= 220;	(*Max position for down movement*)
END_VAR
(*Simulate axis*)
IF NOT bEnable THEN
	iState_Lift := 0;
END_IF;

(*Initialisation*)
IF NOT bInitDone THEN
	(*Randomize system's starting position*)
	lastRandom := RDM(lastRandom);
	fLift_CurrentPos := -100 * lastRandom + 10;
	lastRandom := RDM(lastRandom);
	fPos_angle := 100 * lastRandom + 40; (* X2 = (180 - 100[=X1]) / 2 *)
	bInitDone:=TRUE;
END_IF;

CASE iState_Lift OF
0:	(*Off*)
	IF bEnable THEN
		iState_Lift := 1;
	ELSE
		bLift_InTarget := FALSE;
	END_IF;

1:	(*IDLE*)
	IF bLift_Start THEN
		bLift_InTarget := FALSE;
		iState_Lift := 2;
	END_IF;

2:	(*MovingToTarget*)
	bLift_InTarget := FALSE;
	IF fLift_TargetPos > fLift_CurrentPos THEN
		(*Moving up*)
		fLift_CurrentPos := fLift_CurrentPos + ABS(fLift_Velo);
	ELSIF fLift_TargetPos < fLift_CurrentPos THEN
		(*Moving down*)
		fLift_CurrentPos := fLift_CurrentPos - ABS(fLift_Velo);
	END_IF;
	(*Limit output*)
	fLift_CurrentPos := LIMIT(-220, fLift_CurrentPos, 10);
	(* Moved close to target*)
	IF (ABS(fLift_CurrentPos - fLift_TargetPos) <= ABS(fLift_Velo) ) THEN
		fLift_CurrentPos := fLift_TargetPos;
		iState_Lift := 3;
	END_IF;
	(*Start has been removed*)
	IF NOT bLift_Start THEN
		iState_Lift := 1;
	END_IF;

3:	(*In target*)
	bLift_InTarget := TRUE;
	IF NOT bLift_Start THEN
		iState_Lift := 1;
	END_IF;

ELSE	(*Error / to Default*)
	iState_Lift := 0;
END_CASE;

fPos_Y := -fLift_CurrentPos;


(*Simulate Beam turning*)
IF bBeam_Left AND (fPos_angle > 0) AND NOT bBeam_Right THEN
	fPos_angle := LIMIT(0, (fPos_angle - 15), 180);
END_IF;
IF bBeam_Right AND (fPos_angle < 180) AND NOT bBeam_Left THEN
	fPos_angle := LIMIT(0, (fPos_angle + 15), 180);
END_IF;


(*Calculate visualisation positions for lift and beam*)
fPos_X := -iBEAM_LENGTH*COS(3.1415926535897932384626433832795/180*fPos_angle);
(*fPos_Y := fPos_height;*)
fBasePos_Y := fPos_Y;	(*Used for animations as base position*)

(*Calculate endpositions of the visualisation for the beam*)
IF (fPos_X > 0) THEN
	fPos_Beam_L := 0;
	fPos_Beam_R := fPos_X;
ELSE
	fPos_Beam_L := fPos_X;
	fPos_Beam_R := 0;
END_IF;

(*define finger positions*)
IF bGripper_Close THEN
	fPosFingerDiff := 0;
ELSE
	fPosFingerDiff := 10;
END_IF;

(*Set sensor values*)
(*Set output values*)
bLimit_Top := (fPos_Y <= 0);
bLimit_Bottom := (fPos_Y >= 210);
bHome_Sensor := (fPos_Y <= 5) AND (fPos_Y >= -5);

bBeamAtLeft := (fPos_angle <= 0);
bBeamAtRight := (fPos_angle >= 180);

bGripperIsOpen := NOT bGripper_Close;
bGripperClosed := bGripper_Close;
END_FUNCTION_BLOCK

(* POU Simulation/RDM_From_OSCAT/RDM, ST *)
FUNCTION RDM : REAL
VAR_INPUT
	last : REAL;
END_VAR
VAR
	tn : DWORD;
	tc : INT;
END_VAR
(*
FROM OSCAT 333
version 1.9	10. mar. 2009
programmer 	hugo
tested by		tobias

this function calculates a pseudo random number
to generate the number it reads the sps timer and calculates a random number between 0 and 1:
in order to use rdm more then once within one sps cycle it need to be called with different seed numbers LAST.

*)
tn := T_PLC_MS();
tc := BIT_COUNT(tn);
tn.31 := tn.2;
tn.30 := tn.5;
tn.29 := tn.4;
tn.28 := tn.1;
tn.27 := tn.0;
tn.26 := tn.7;
tn.25 := tn.6;
tn.24 := tn.3;
tn := ROL(tn,BIT_COUNT(tn)) OR 16#80000001;
tn := tn MOD 71474513 + INT_TO_DWORD(tc + 77);
RDM := FRACT(DWORD_TO_REAL(tn) / 10000000.0 * (math.E - LIMIT(0.0,last,1.0)));


(*
pt := ADR(temp);
pt^ := (T_PLC_MS() AND 16#007FFFFF) OR 16#3D000000;
RDM := fract(modR(temp*e+pi1, PI1-last) + modR(temp*PI1+e + last,e-last));
*)

(* revision history
hm		16. jan 2007		rev 1.0
	original version

hm		11. nov 2007		rev 1.1
	changed time() into t_plc_ms()

hm		20. nov 2007		rev 1.2
	changed code of temp calculation to avoid overflow in modr due to resuclt would not fit DINT for high timeer values

hm		5. jan 2008		rev 1.3
	changed calculation of temp to avoid problem with high values of t_plc_ms

hm		2. feb 2008		rev 1.4
	changed algorithm to avoind non iec functions and guarantee more randomness

hm	10. mar. 2008		rev 1.5
	make sure last will be between 0 and 1 to avoid invalid results

hm	16. mar. 2008		rev 1.6
	added conversion for tc to avoid warnings under codesys 3.0

hm	18. may. 2008		rev 1.7
	changed constant E to E1

hm	18. oct. 2008		rev 1.8
	using math constants

hm	10. mar. 2009		rev 1.9
	real constants updated to new systax using dot

*)
END_FUNCTION

(* POU Simulation/RDM_From_OSCAT/T_PLC_MS, ST *)
FUNCTION T_PLC_MS : DWORD
VAR CONSTANT
	debug : BOOL := 0;
	N : INT := 0;
	offset : DWORD := 0;
END_VAR
VAR
	tx : TIME;
END_VAR
(*
	From OSCAT 333
	version 1.2	16. nov 2008
	programmer 	hugo
	tested BY	oscat

	T_PLC_MS reads the internal PLC timer AND RETURN the TIME, it has the advantage TO be able TO set a debug mode
AND SPEED up the counter TO test the plc timer overrun which occurs every 50 days respectively 25 days AT siemens S7
	this routine also allows TO correct the behavior OF s7 where the internal plc counter will NOT count all 32 bits.
*)
tx := TIME();
T_PLC_MS := TIME_TO_DWORD(Tx);
(* hier muss die korrektur für step7 stattfinden
plctime muss den vollen wertebereich von time ausnutzen:
wenn bei step7 time -24tage bis plus 24 tage ist dann muss der timer auch beim überlauf auf -24tage springen 
und auf keinen fall auf 0 !!!!
für siemens muss ein weiterer fb im main eingebunden werden der sicherstellt das alle 32 bits durchgezählt werden.
es kann nur ein fb sein den er muss sich das oberste (32te) bit merken.
oder etwa spring s7 bei überlauf auf -24 tage????? dann wäre keine korrektur nötig.
*)
IF debug THEN
	T_PLC_MS := (SHL(T_PLC_MS,N) OR SHL(DWORD#1,N)-1) + OFFSET;
END_IF;

(* revision history
hm	14.9.2007	rev 1.0
	original version

hm	12. nov 2007	rev 1.1
	added temporaray variable tx because some compilers could not handle time() as an argument

hm	16. nov. 2008	rev 1.2
	initialized constants with 0 for compatibility reasons
*)
END_FUNCTION

(* POU Simulation/RDM_From_OSCAT/BIT_COUNT, ST *)
FUNCTION BIT_COUNT : INT
VAR_INPUT
	IN : DWORD;
END_VAR
VAR
END_VAR
(*
OSCAT 333
version 1.1	10 sep 2007
programmer 	hugo
tested by		tobias

BIT_COUNT counts the amount True of bits in a dword.
for exabple: bit_count(3) returns 2 because two bits (bits 0 and 1) are true and all others are false. 
*)
WHILE in > 0 DO
	IF in.0 THEN Bit_Count := Bit_Count + 1; END_IF;
	in := SHR(in,1);
END_WHILE;



(* revision history
5.7.2007	rev 1.0		original version

10.9.2007	rev 1.1		hm
	changed algorithm for better performace
	the execution time has reduced by a factor of 5
	deleted unused variable temp
*)
END_FUNCTION

(* POU Simulation/RDM_From_OSCAT/FRACT, ST *)
FUNCTION FRACT : REAL
VAR_INPUT
	x : REAL;
END_VAR
VAR
END_VAR
(*
From OSCAT 333
version 1.3	10. mar. 2009
programmer 	hugo
tested by		tobias

this function returns the fraction of a real number
fract(3.14) = 0.14

*)
IF ABS(x) < 2.0E9 THEN
	FRACT := x - DINT_TO_REAL(D_TRUNC(x));
ELSE
	FRACT := 0.0;
END_IF;

(* revision history
hm	4. aug 2006	rev 1.0
	original version

hm	11. mar 2008	rev 1.1
	added dint_to_real for compatibility reasons
	now returns 0 for number > 2e9
	changed input to x

hm	21. mar. 2008	rev 1.2
	use D_trunc instead of TRUNC for compatibility reasons

hm	10. mar. 2009	rev 1.3
	real constants updated to new systax using dot

*)
END_FUNCTION

(* POU Simulation/RDM_From_OSCAT/D_TRUNC, ST *)
FUNCTION D_TRUNC : DINT
VAR_INPUT
	X : REAL;
END_VAR
VAR
END_VAR
(*
From OSCAT 333
version 1.2	10. mar. 2009
programmer 	hugo
tested by		oscat

d_trunc truncates a real to a dint 1.5 will be 1 and -1.5 will be -1
d_trunc is necessary because many systems do not offer a trunc to a dint
also real_to_dint will not deliver the same result on different systems

*)
D_TRUNC := REAL_TO_DINT(X);
IF X > 0.0 THEN
	IF DINT_TO_REAL(D_TRUNC) > X THEN D_TRUNC := D_TRUNC - 1; END_IF;
ELSE
	IF DINT_TO_REAL(D_TRUNC) < X THEN D_TRUNC := D_TRUNC + 1; END_IF;
END_IF;


(* for systems that support a dint truncation this routine can be replaced by trunc() *)


(* revision history
hm	21. mar. 2008	rev 1.0
	original version

hm	31. oct. 2008	rev 1.1
	optimized performance

hm	10. mar. 2009	rev 1.2
	real constants updated to new systax using dot
*)
END_FUNCTION

(* POU Simulation/FB_Simu_Drill, ST *)
FUNCTION_BLOCK FB_Simu_Drill
(*Simulation model for the behaviour of the Drill machine.
Author: Niko Siltala, niko.siltala@tut.fi, Tampere University of Technology / MEI
Date: 2016-12-12
Version: 1.0
*)
VAR_INPUT
	bEnable			: BOOL := TRUE;	(*Enable drill*)
	bLift_Start		: BOOL;		(*Triggers and starts the lift movement at rising edge*)
	fLift_Velo		: REAL := 10;	(*Velocity*)
	fLift_TargetPos	: REAL;		(*Target position*)
	bDrillOn			: BOOL;		(*Drill is On*)
	bFixture_Close	: BOOL; 	(*Close Fixture*)
	bInitDone		: BOOL;		(*Initialisation done for simulated machine*)
END_VAR
VAR_OUTPUT
	bLift_InTarget	: BOOL;	(*Lift has reached the target*)
	fLift_CurrentPos	: REAL;	(*Current position of the lift*)
	bLimit_Top		: BOOL;	(*Height position at top limit*)
	bLimit_Bottom	: BOOL;	(*Height position at bottom limit*)
	bHome_Sensor	: BOOL;	(*Height position at home limit*)
	bFixture_Open	: BOOL;	(*Fixture is Open*)
	bFixture_Closed	: BOOL;	(*Fixture is Closed*)
END_VAR
VAR_IN_OUT
	stPart_inFixture : ST_Part; 	(*Data structure for the part*)
END_VAR
VAR
	fPos_height	: REAL;	(* Manipulators height position*)
	fPos_Y		: REAL;	(* Manipulator's Y position*)
	fBasePos_Y 	: REAL; (*Position of manipulator base*)
	iState_Lift	: UINT;	(*State of beam model*)
	iRPMCurrent	: INT;	(*Current RPM*)
	fPosJawDiff 	: REAL;	(*Right fixture jaw position. 0 position when grasping.*)
END_VAR
VAR CONSTANT
	fPOS_MAX_DOWN		: REAL	:= 170;	(*Max position for down movement*)
	iSPINDLE_RPM_MAX	: INT	:= 600;	(*Max RPM for Spindle*)
END_VAR
(*Simulate axis*)
IF NOT bEnable THEN
	iState_Lift := 0;
END_IF;

(*Initialisation*)
IF NOT bInitDone THEN
	(*Randomize system's starting position*)
	lastRandom := RDM(lastRandom);
	fLift_CurrentPos := -60 * lastRandom + 10;
	bInitDone:=TRUE;
END_IF;

CASE iState_Lift OF
0:	(*Off*)
	IF bEnable THEN
		iState_Lift := 1;
	ELSE
		bLift_InTarget := FALSE;
	END_IF;

1:	(*IDLE*)
	IF bLift_Start THEN
		bLift_InTarget := FALSE;
		iState_Lift := 2;
	END_IF;

2:	(*MovingToTarget*)
	bLift_InTarget := FALSE;
	IF fLift_TargetPos > fLift_CurrentPos THEN
		(*Moving up*)
		fLift_CurrentPos := fLift_CurrentPos + ABS(fLift_Velo);
	ELSIF fLift_TargetPos < fLift_CurrentPos THEN
		(*Moving down*)
		fLift_CurrentPos := fLift_CurrentPos - ABS(fLift_Velo);
	END_IF;
	(*Limit output*)
	fLift_CurrentPos := LIMIT(-fPOS_MAX_DOWN, fLift_CurrentPos, 10);
	(* Moved close to target*)
	IF (ABS(fLift_CurrentPos - fLift_TargetPos) <= ABS(fLift_Velo) ) THEN
		fLift_CurrentPos := fLift_TargetPos;
		iState_Lift := 3;
	END_IF;
	(*Start has been removed*)
	IF NOT bLift_Start THEN
		iState_Lift := 1;
	END_IF;

3:	(*In target*)
	bLift_InTarget := TRUE;
	IF NOT bLift_Start THEN
		iState_Lift := 1;
	END_IF;

ELSE	(*Error / to Default*)
	iState_Lift := 0;
END_CASE;

fPos_Y := -fLift_CurrentPos;
fBasePos_Y := fPos_Y;	(*Used for animations as base position*)


(*define fixture jaws positions*)
IF bFixture_Close THEN
	fPosJawDiff := 0;
ELSE
	fPosJawDiff := 10;
END_IF;

(*Set sensor values*)
(*Set output values*)
bLimit_Top := (fPos_Y <= 0);
bLimit_Bottom := (fPos_Y >= (fPOS_MAX_DOWN-10));
bHome_Sensor := (fPos_Y <= 5) AND (fPos_Y >= -5);

bFixture_Open := NOT bFixture_Close;
bFixture_Closed := bFixture_Close;

IF bDrillOn THEN
	iRPMCurrent := iRPMCurrent + 100;
ELSE
	iRPMCurrent := iRPMCurrent - 20;
END_IF;
iRPMCurrent := LIMIT(0, iRPMCurrent, iSPINDLE_RPM_MAX);
END_FUNCTION_BLOCK

(* POU Simulation/F_MovePartForward, ST *)
FUNCTION F_MovePartForward : BOOL
(*Moves parts forward on conveyour, if possible*)
VAR_INPUT
END_VAR
VAR_IN_OUT
	arrParts : ARRAY [0..10] OF ST_Part;	(*Array of parts*)
END_VAR
VAR
	i : INT;	(*indexer*)
	j : INT;	(*indexer*)
END_VAR
(*Moves parts forward as much there is free places*)
FOR i:= 0 TO 9 DO
	j := i +1;
	IF NOT arrParts[i].bExists THEN
		IF arrParts[j].bExists THEN
			F_CopyPart(arrParts[j], arrParts[i]);
			arrParts[j].bExists := FALSE;
			arrParts[j].bHasHole := FALSE;
		END_IF;
	END_IF;
END_FOR;

F_MovePartForward := TRUE;
END_FUNCTION

(* POU Simulation/F_CopyPart, ST *)
FUNCTION F_CopyPart : BOOL
(*Moves part data from part to part*)
VAR_INPUT
END_VAR
VAR_IN_OUT
	stPartFrom : ST_Part;	(*The copied part - From*)
	stPartTo : ST_Part;	(*Where to copy the part*)
END_VAR
VAR
END_VAR
(*Moves part data from part to part*)
stPartTo.bExists := stPartFrom.bExists;
stPartTo.bHasHole := stPartFrom.bHasHole;
stPartTo.posX := stPartFrom.posX;
stPartTo.posY := stPartFrom.posY;

F_CopyPart:=TRUE;
END_FUNCTION

(* POU Examples/PRG_SFC_Example, SFC *)
PROGRAM PRG_SFC_Example
VAR_INPUT
	bReset		: BOOL;	(*Reset Request*)
END_VAR
VAR_OUTPUT
END_VAR
VAR
	bLocalReset	: BOOL;	(*Performs local reset*)
	SFCReset 	: BOOL;	(*Resets the execution of SFC to init once this SFCFlag is set true *)
END_VAR
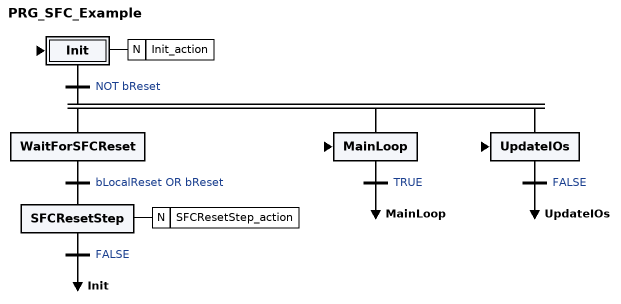
INITIAL_STEP Init:
	Init_action(N);
END_STEP
TRANSITION FROM Init TO (WaitForSFCReset, MainLoop, UpdateIOs) := NOT bReset;
END_TRANSITION
STEP WaitForSFCReset:
END_STEP
TRANSITION FROM WaitForSFCReset TO SFCResetStep := bLocalReset OR bReset;
END_TRANSITION
STEP SFCResetStep:
	SFCResetStep_action(N);
END_STEP
TRANSITION FROM SFCResetStep TO Init := FALSE;
END_TRANSITION
STEP MainLoop:
END_STEP
TRANSITION FROM MainLoop TO MainLoop := TRUE;
END_TRANSITION
STEP UpdateIOs:
END_STEP
TRANSITION FROM UpdateIOs TO UpdateIOs := FALSE;
END_TRANSITION

ACTION Init_action:
SFCReset := FALSE;
bLocalReset	:= FALSE;
END_ACTION

ACTION SFCResetStep_action:
SFCReset := TRUE;
END_ACTION
END_PROGRAM

(* Visualisation Simulator/Components/VC_Beacon
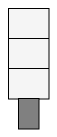
rectangle at (0,0)-(41,31): alarm colour if $red$
rectangle at (0,30)-(41,61): alarm colour if $yellow$
rectangle at (0,60)-(41,91): alarm colour if $green$
1 more shapes without text or variables
*)

(* Visualisation Simulator/ErrorPanels/VC_ErrorDetail_Drill
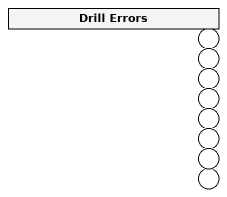
embedded screen at (0,20)-(211,41): VC_ErrorItem
rectangle at (0,0)-(211,21): text "Drill Errors"
embedded screen at (0,40)-(211,61): VC_ErrorItem
embedded screen at (0,160)-(211,181): VC_ErrorItem
embedded screen at (0,60)-(211,81): VC_ErrorItem
embedded screen at (0,80)-(211,101): VC_ErrorItem
embedded screen at (0,100)-(211,121): VC_ErrorItem
embedded screen at (0,120)-(211,141): VC_ErrorItem
embedded screen at (0,140)-(211,161): VC_ErrorItem
*)

(* Visualisation Simulator/ErrorPanels/VC_ErrorDetail_Manip
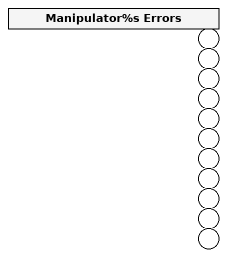
embedded screen at (0,20)-(211,41): VC_ErrorItem
rectangle at (0,0)-(211,21): text "Manipulator%s Errors"; shows $manipName$
embedded screen at (0,40)-(211,61): VC_ErrorItem
embedded screen at (0,60)-(211,81): VC_ErrorItem
embedded screen at (0,80)-(211,101): VC_ErrorItem
embedded screen at (0,80)-(211,101): VC_ErrorItem
embedded screen at (0,100)-(211,121): VC_ErrorItem
embedded screen at (0,120)-(211,141): VC_ErrorItem
embedded screen at (0,140)-(211,161): VC_ErrorItem
embedded screen at (0,160)-(211,181): VC_ErrorItem
embedded screen at (0,180)-(211,201): VC_ErrorItem
embedded screen at (0,200)-(211,221): VC_ErrorItem
embedded screen at (0,220)-(211,241): VC_ErrorItem
*)

(* Visualisation Simulator/VC_ErrorDetails
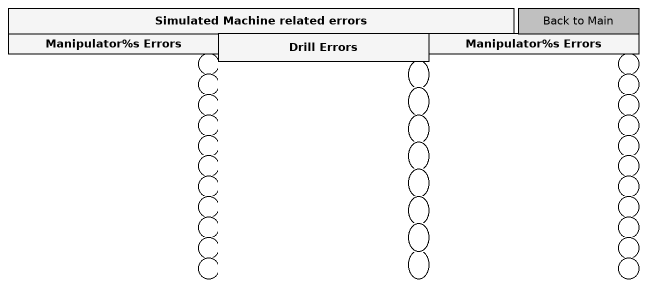
embedded screen at (0,25)-(211,271): VC_ErrorDetail_Manip
rectangle at (0,0)-(506,26): text "Simulated Machine related errors"
embedded screen at (420,25)-(631,271): VC_ErrorDetail_Manip
embedded screen at (210,25)-(421,271): VC_ErrorDetail_Drill
rounded rectangle at (510,0)-(631,26): text "Back to Main"; opens VISU_SimulatedMachine
*)

(* Visualisation Simulator/Components/VC_ErrorItem
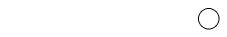
rectangle at (0,0)-(191,21): text "%s :"; shows $name$; alarm colour if $flag$
ellipse at (190,0)-(211,21): alarm colour if $flag$
1 more shapes without text or variables
*)

(* Visualisation Simulator/FBs/VC_FB_Simu_Drill
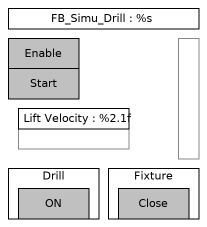
rectangle at (100,160)-(191,211): text "Fixture"
rectangle at (0,160)-(91,211): text "Drill"
rounded rectangle at (0,30)-(71,61): text "Enable"; alarm colour if $FB$.bEnable; toggles $FB$.bEnable
rectangle at (0,0)-(191,21): text "FB_Simu_Drill : %s"; shows $Name$
rounded rectangle at (0,60)-(71,91): text "Start"; alarm colour if $FB$.bLift_Start; taps $FB$.bLift_Start
rectangle at (10,100)-(121,121): text "Lift Velocity : %2.1f"; shows $FB$.fLift_Velo
rounded rectangle at (10,180)-(81,211): text "ON"; alarm colour if $FB$.bDrillOn; toggles $FB$.bDrillOn
rounded rectangle at (110,180)-(181,211): text "Close"; alarm colour if $FB$.bFixture_Close; toggles $FB$.bFixture_Close
2 more shapes without text or variables
1 elements of other kinds (tables, trends, ...) not read
*)

(* Visualisation Simulator/FBs/VC_FB_Simu_Manipulator
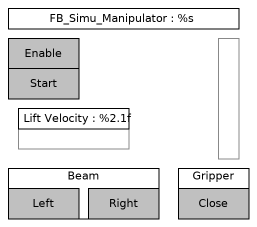
rectangle at (170,160)-(241,211): text "Gripper"
rectangle at (0,160)-(151,211): text "Beam"
rounded rectangle at (0,30)-(71,61): text "Enable"; alarm colour if $FB$.bEnable; toggles $FB$.bEnable
rectangle at (0,0)-(231,21): text "FB_Simu_Manipulator : %s"; shows $Name$
rounded rectangle at (0,60)-(71,91): text "Start"; alarm colour if $FB$.bLift_Start; taps $FB$.bLift_Start
rectangle at (10,100)-(121,121): text "Lift Velocity : %2.1f"; shows $FB$.fLift_Velo
rounded rectangle at (0,180)-(71,211): text "Left"; alarm colour if $FB$.bBeam_Left; toggles $FB$.bBeam_Left
rounded rectangle at (80,180)-(151,211): text "Right"; alarm colour if $FB$.bBeam_Right; toggles $FB$.bBeam_Right
rounded rectangle at (170,180)-(241,211): text "Close"; alarm colour if $FB$.bGripper_Close; toggles $FB$.bGripper_Close
2 more shapes without text or variables
1 elements of other kinds (tables, trends, ...) not read
*)

(* Visualisation Simulator/MachineComponents/VC_Panel_MachineControl
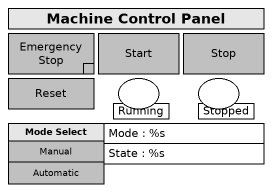
rounded rectangle at (0,25)-(86,66): text "Emergency / Stop"; alarm colour if PRG_Simulator.bBtn_EmergencyStop; toggles PRG_Simulator.bBtn_EmergencyStop
rounded rectangle at (90,25)-(171,66): text "Start"; alarm colour if .I_Btn_Start; taps .I_Btn_Start
rounded rectangle at (0,70)-(86,101): text "Reset"; alarm colour if .I_Btn_Reset; taps .I_Btn_Reset
rounded rectangle at (175,25)-(256,66): text "Stop"; alarm colour if .I_Btn_Stop; taps .I_Btn_Stop
rectangle at (0,0)-(256,21): text "Machine Control Panel"
rectangle at (95,115)-(256,136): text "Mode : %s"; shows .fbStateModel.eMode
rectangle at (95,135)-(256,156): text "State : %s"; shows .fbStateModel.eState
embedded screen at (0,115)-(96,176): VC_Panel_ModeSelector
rectangle at (105,95)-(161,111): text "Running"
rectangle at (190,95)-(246,111): text "Stopped"
ellipse at (110,70)-(151,101): alarm colour if .O_Light_Start
ellipse at (190,70)-(231,101): alarm colour if .O_Light_Stop
embedded screen at (75,55)-(86,66): VC_sensor
*)

(* Visualisation Simulator/MachineComponents/VC_Panel_ModeSelector
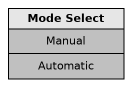
rounded rectangle at (0,20)-(116,46): text "Manual"; alarm colour if .HMI_uModeReq=3; runs INTERN ASSIGN HMI_uModeReq:=(3)
rectangle at (0,0)-(116,21): text "Mode Select"
rounded rectangle at (0,45)-(116,71): text "Automatic"; alarm colour if .HMI_uModeReq=1; runs INTERN ASSIGN HMI_uModeReq:=(1)
*)

(* Visualisation Simulator/Components/VC_Part
rectangle at (0,0)-(41,51): invisible if NOT $part$.bExists
rectangle at (15,0)-(26,41): invisible if NOT $part$.bExists OR NOT $part$.bHasHole
*)

(* Visualisation Simulator/Components/VC_sensor
rectangle at (0,0)-(11,11): alarm colour if $VAR$
*)

(* Visualisation Simulator/MachineComponents/VC_Simu_Conv_In
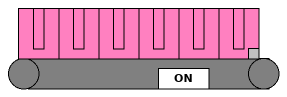
embedded screen at (210,0)-(251,51): VC_Part
embedded screen at (240,40)-(251,51): VC_sensor
embedded screen at (170,0)-(211,51): VC_Part
embedded screen at (130,0)-(171,51): VC_Part
embedded screen at (90,0)-(131,51): VC_Part
embedded screen at (50,0)-(91,51): VC_Part
embedded screen at (10,0)-(51,51): VC_Part
rectangle at (150,60)-(201,81): text "OFF"
rectangle at (150,60)-(201,81): text "ON"; invisible if NOT $MotOn$
3 more shapes without text or variables
*)

(* Visualisation Simulator/MachineComponents/VC_Simu_Drill
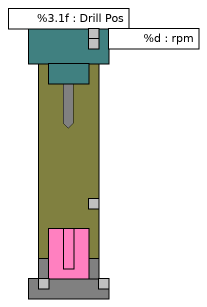
rectangle at (20,20)-(101,56): y offset $FB$.fBasePos_Y
rectangle at (0,0)-(121,21): text "%3.1f : Drill Pos"; shows $FB$.fLift_CurrentPos
embedded screen at (80,20)-(91,31): VC_sensor
embedded screen at (80,190)-(91,201): VC_sensor
embedded screen at (80,30)-(91,41): VC_sensor
polygon at (55,75)-(65,120): alarm colour if $FB$.iRPMCurrent > 0; y offset $FB$.fBasePos_Y
rectangle at (40,55)-(81,76): y offset $FB$.fBasePos_Y
rectangle at (30,250)-(41,271): x offset - $FB$.fPosJawDiff
rectangle at (80,250)-(91,271): x offset $FB$.fPosJawDiff
embedded screen at (40,220)-(81,271): VC_Part
embedded screen at (90,270)-(101,281): VC_sensor
embedded screen at (30,270)-(41,281): VC_sensor
rectangle at (100,20)-(191,41): text "%d : rpm"; shows $FB$.iRPMCurrent
2 more shapes without text or variables
*)

(* Visualisation Simulator/MachineComponents/VC_Simu_Manipulator
